// TwinCAT 3 PLC project X881_Booth_Esclave
// libraries:
//   CmpBitmapPool, * (System)
//   Tc2_Standard, * (Beckhoff Automation GmbH)
//   Tc2_SUPS, * (Beckhoff Automation GmbH)
//   Tc2_System, * (Beckhoff Automation GmbH)
//   Tc2_Utilities, * (Beckhoff Automation GmbH)
//   Tc3_Module, * (Beckhoff Automation GmbH)
//   VisuDialogs, * (System)
//   BASIC,3.3.3.0,OSCAT
//   Tc2_ModbusRTU,3.6.1.0,Beckhoff Automation GmbH
//   Tc2_SerialCom,3.4.6.0,Beckhoff Automation GmbH
//   Tc2_SystemCX,3.5.3.0,Beckhoff Automation GmbH
//   Tc2_TcpIp,3.4.2.0,Beckhoff Automation GmbH
//   Util,3.5.11.0,System
//   VisuSymbols,3.5.10.0,System
// project tree:
//   Data types/Autres/ ST_Alarmes.TcDUT
//   Data types/Com_IP/ E_ClientSteps.TcDUT, E_DataExchaSteps.TcDUT, E_ServerSteps.TcDUT
//   Data types/Objets/ Objet_BatElec.TcDUT, Objet_Moteur_EC.TcDUT, Objet_Mot_TOR.TcDUT, Objet_Pressostat.TcDUT, Objet_Registre.TcDUT, Objet_RegulPI.TcDUT, Objet_Sonde.TcDUT
//   Global Variables/ Global_Variables.TcGVL, GVL_RegTROX.TcGVL, GVL_Visu.TcGVL, Variable_Configuration.TcGVL
//   / GlobalTextList.TcGTLO, Recipe Manager.TcRMO (not stored), Standard.TcTTO, Tache_test.TcTTO, Visualization Manager.TcVMO (not stored), VISU_TASK.TcTTO
//   POUs/ a1_MAIN.TcPOU, a2_Gestion_ES.TcPOU, a3_Ecriture_Bit.TcPOU, a4_Lecture_Bit.TcPOU, a5_Ecriture_InterCom.TcPOU, a6_Lecture_InterCom.TcPOU, b_SCL_Mesures.TcPOU, c_Gestion_Defaut.TcPOU, d_Gestion_Pause_Modes.TcPOU, e_Gestion_Horraire.TcPOU, f_Gestion_Etats.TcPOU, g_Gestion_Texte_Modes.TcPOU, h_Enr_Recette.TcPOU, i_Protocol_Auto.TcPOU, j_Protocol_Manu.TcPOU, l_Cons_LED.TcPOU, n0_Regulation_Bas_Deb.TcPOU, n1_Regulation_Press.TcPOU, n2_Regulation_Temp.TcPOU, n3_Regul_Temp_EauMitig.TcPOU, o_Cons_Cmd_Actionneurs.TcPOU, p_Com_Modbus_RS485.TcPOU, q_Gestion_Actionneurs_ANA.TcPOU, r_Gestion_Actionneurs_TOR.TcPOU, s_InterCom_Esclave.TcPOU, t_Enr_Variables.TcPOU
//   POUs/Block/Autres/ Blinck_V2.TcPOU, Dew_Point.TcPOU, Filtre_V1.TcPOU, Prise.TcPOU, PWM.TcPOU, RTC_Time.TcPOU, SCL.TcPOU, SCL_Real.TcPOU, Sontay_4RM.TcPOU, TON_V1.TcPOU, UP_DOWN_RATE.TcPOU
//   POUs/Block/Cabines/ Com485_Dalcnet.TcPOU, Com485_RegTROX.TcPOU, Gache.TcPOU, Humidificateur.TcPOU, Integr_Vol_Eau.TcPOU, Mode.TcPOU, Registre_V1.TcPOU, Servomoteur_V1.TcPOU
//   POUs/Block/Com_Ip/ FB_LocalServer.TcPOU, FB_RemoteClient.TcPOU, FB_ServerDataExcha.TcPOU, LogError.TcPOU, LogMessage.TcPOU, SCODE_CODE.TcPOU
//   POUs/Block/Objets/ BatElec.TcPOU, Moteur_EC.TcPOU, Objet_Mot_TOR_V1.TcPOU, Objet_PI_V1.TcPOU, Objet_Pressostat_V1.TcPOU, Objet_Registre_V1.TcPOU, Objet_Sonde_V1.TcPOU
//   POUs/Gestion_Enceinte_Clim/ B_Gestion_Defaut.TcPOU, C0_Gestion_Consignes.TcPOU, C_Regul_Temp.TcPOU, D_Regul_Humi.TcPOU, E_Cons_Cmd_Actionneurs.TcPOU, F_Gestion_Actionneurs.TcPOU
//   POUs/Visualisation/ Alarmes.TcPOU, Visu.TcPOU
//   Visualizations/Visualizations/ Accueil.TcVIS, Depollution.TcVIS, Maintenance_2.TcVIS, Maintenance_3.TcVIS, Maintenance_4.TcVIS, Maintenance_5.TcVIS, Maintenance_6.TcVIS, Maintenance_7.TcVIS, ModeManuel.TcVIS, Nettoyage.TcVIS, Maintenance_1.TcVIS, menu.TcVIS, Recet_EnCours.TcVIS, Sel_Recettes.TcVIS
//   Visualizations/Visualizations/Fonds/ masque.TcVIS
//   Visualizations/Visualizations/GestionAlarme/Programme/ GestionAlarme.TcPOU
//   Visualizations/Visualizations/GestionAlarme/Structures/ Erreur_Struct.TcDUT, Erreur_StructVisu.TcDUT
//   Visualizations/Visualizations/Images/ ImagePool_Clean.TcIPO (not stored), ImagePool.TcIPO (not stored), ImagePool_Action.TcIPO (not stored), ImagePool_Buttons.TcIPO (not stored)
//   Visualizations/Visualizations/Mes_Textes/ Noms_Modes.TcTLO, Etats_Cabine.TcTLO
//   Visualizations/Visualizations/Objets/ Door.TcVIS, Sink.TcVIS, Drain.TcVIS, Plug.TcVIS
//   Visualizations/Visualizations/PopUp/ Actionneurs.TcVIS, Alarmes.TcVIS, PopUp_Alarms.TcVIS, PopUp_Hight_Level.TcVIS
// real-time tasks:
//   TASK Standard: cycle T#20ms, priority 8, ADS port 350
//   TASK Tache_test: cycle T#10ms, priority 6, ADS port 351
//   TASK VISU_TASK: cycle T#100000us, priority 10, ADS port 352
// I/O:
//   DEVICE Périphérique 2 (EtherCAT), AmsNetId 5.138.94.134.3.1
//     Terme 1 (EK1200) [EK1200-5000 EtherCAT Power supply (2A E-Bus)]
//       Terme 2 (EL1809) [EL1809 16Ch. Dig. Input 24V, 3ms]
//       Terme 3 (EL2828) [EL2828 8Ch. Dig. Output 24V, 2A]
//       Terme 4 (EL3068) [EL3068 8Ch. Ana. Input 0-10V]
//       Terme 5 (EL4008) [EL4008 8Ch. Ana. Output 0-10V, 12bit]
//       Terme 6 (EL6021) [EL6021 Interface (RS422/485)]
//       Terme 7 (EL3068) [EL3068 8Ch. Ana. Input 0-10V]
//       Terme 8 (EL9011) [EL9011 End Terminal]
// variable links:
//   X881_Booth_Esclave/X881_Booth_Esclave Instance <-> Device 2 (EtherCAT)/Term 1 (EK1200)/Term 2 (EL1809)
//     Standard Inputs/Global_Variables.ETOR10_Hygrostat_Souf_CT <-> Channel 10/Input
//     Standard Inputs/Global_Variables.ETOR11_Pressostat_Secu <-> Channel 11/Input
//     Standard Inputs/Global_Variables.ETOR12_Thermostat_Secu <-> Channel 12/Input
//     Standard Inputs/Global_Variables.ETOR13_Marche_BatElec_CTA <-> Channel 13/Input
//     Standard Inputs/Global_Variables.ETOR14_Libre <-> Channel 14/Input
//     Standard Inputs/Global_Variables.ETOR15_Libre <-> Channel 15/Input
//     Standard Inputs/Global_Variables.ETOR16_Libre <-> Channel 16/Input
//     Standard Inputs/Global_Variables.ETOR1_Fdc_Va_Vid_Lavabo_Ouv <-> Channel 1/Input
//     Standard Inputs/Global_Variables.ETOR2_Fdc_Va_Vid_Lavabo_Ferm <-> Channel 2/Input
//     Standard Inputs/Global_Variables.ETOR3_Info_Ma_Prise <-> Channel 3/Input
//     Standard Inputs/Global_Variables.ETOR4_Service_Humi_CTA <-> Channel 4/Input
//     Standard Inputs/Global_Variables.ETOR5_Def_Humi_CTA <-> Channel 5/Input
//     Standard Inputs/Global_Variables.ETOR6_Info_Contact_Porte <-> Channel 6/Input
//     Standard Inputs/Global_Variables.ETOR7_Def_MotRep_Souf_CTA <-> Channel 7/Input
//     Standard Inputs/Global_Variables.ETOR8_Def_MotSouf_Souf_CTA <-> Channel 8/Input
//     Standard Inputs/Global_Variables.ETOR9_Def_Alim_BatElec_CTA <-> Channel 9/Input
//   X881_Booth_Esclave/X881_Booth_Esclave Instance <-> Device 2 (EtherCAT)/Term 1 (EK1200)/Term 3 (EL2828)
//     Standard Outputs/Global_Variables.STOR1_Cmd_EV_Alim_Lavabo <-> Channel 1/Output
//     Standard Outputs/Global_Variables.STOR2_Cmd_Va_Vid_Lavabo <-> Channel 2/Output
//     Standard Outputs/Global_Variables.STOR3_Cmd_Ma_Prise <-> Channel 3/Output
//     Standard Outputs/Global_Variables.STOR4_Cmd_BatElec_CTA <-> Channel 4/Output
//     Standard Outputs/Global_Variables.STOR{5..8}_Libre <-> Channel {5..8}/Output  (4 links)
//   X881_Booth_Esclave/X881_Booth_Esclave Instance <-> Device 2 (EtherCAT)/Term 1 (EK1200)/Term 4 (EL3068)
//     Standard Inputs/Global_Variables.EAN1_Sonde_Debit_Eau_Lavabo <-> AI Standard Channel 1/Value
//     Standard Inputs/Global_Variables.EAN2_Sonde_Temp_Cabine <-> AI Standard Channel 2/Value
//     Standard Inputs/Global_Variables.EAN3_Sonde_Hygro_Cabine <-> AI Standard Channel 3/Value
//     Standard Inputs/Global_Variables.EAN4_Sonde_Temp_Batt_EG <-> AI Standard Channel 4/Value
//     Standard Inputs/Global_Variables.EAN5_Sonde_Pression_Cabine <-> AI Standard Channel 5/Value
//     Standard Inputs/Global_Variables.EAN6_Sonde_press_Souf <-> AI Standard Channel 6/Value
//     Standard Inputs/Global_Variables.EAN7_Retour_Pos_Reg_Etanche_Ext <-> AI Standard Channel 7/Value
//     Standard Inputs/Global_Variables.EAN8_Sonde_press_Ext <-> AI Standard Channel 8/Value
//   X881_Booth_Esclave/X881_Booth_Esclave Instance <-> Device 2 (EtherCAT)/Term 1 (EK1200)/Term 5 (EL4008)
//     Standard Outputs/Global_Variables.SAN1_Cons_Humi_CTA <-> AO Outputs Channel 1/Analog output
//     Standard Outputs/Global_Variables.SAN2_Cons_MotRep_CTA <-> AO Outputs Channel 2/Analog output
//     Standard Outputs/Global_Variables.SAN3_Cons_MotSouf_CTA <-> AO Outputs Channel 3/Analog output
//     Standard Outputs/Global_Variables.SAN4_Cons_BatElec_CTA <-> AO Outputs Channel 4/Analog output
//     Standard Outputs/Global_Variables.SAN5_Cons_V3V_Froid_CTA <-> AO Outputs Channel 5/Analog output
//     Standard Outputs/Global_Variables.SAN6_Libre <-> AO Outputs Channel 6/Analog output
//     Standard Outputs/Global_Variables.SAN8_Libre <-> AO Outputs Channel 8/Analog output
//     Standard Outputs/Global_Variables.SAN7_Cons_Ouv_Reg_Etanche_Ext <-> AO Outputs Channel 7/Analog output
//   X881_Booth_Esclave/X881_Booth_Esclave Instance <-> Device 2 (EtherCAT)/Term 1 (EK1200)/Term 6 (EL6021)
//     Tache_test Inputs/Global_Variables.MB.InData/D[{0..21}] <-> COM TxPDO-Map Inputs/Data In {0..21}  (22 links)
//     Tache_test Inputs/Global_Variables.MB.InData/Status <-> COM TxPDO-Map Inputs/Status
//     Tache_test Outputs/Global_Variables.MB.OutData/Ctrl <-> COM RxPDO-Map Outputs/Ctrl
//     Tache_test Outputs/Global_Variables.MB.OutData/D[{0..21}] <-> COM RxPDO-Map Outputs/Data Out {0..21}  (22 links)
//   X881_Booth_Esclave/X881_Booth_Esclave Instance <-> Device 2 (EtherCAT)/Term 1 (EK1200)/Term 7 (EL3068)
//     Standard Inputs/Global_Variables.EAN{10..16}_Libre <-> AI Standard Channel {2..8}/Value  (7 links)
//     Standard Inputs/Global_Variables.EAN9_Sonde_Temp_Souf <-> AI Standard Channel 1/Value

CONFIGURATION X881_Booth_Esclave
    RESOURCE PLC ON TwinCAT3
        TASK Standard(INTERVAL := T#20ms, PRIORITY := 8);
        TASK Tache_test(INTERVAL := T#10ms, PRIORITY := 6);
        TASK VISU_TASK(INTERVAL := T#100000us, PRIORITY := 10);
        PROGRAM a1_MAIN WITH Standard : a1_MAIN;
        PROGRAM p_Com_Modbus_RS485 WITH Tache_test : p_Com_Modbus_RS485;
        PROGRAM VisuElems_Visu_Prg WITH VISU_TASK : VisuElems.Visu_Prg;
    END_RESOURCE
END_CONFIGURATION

// ---- Data types/Autres/ST_Alarmes.TcDUT
TYPE ST_Alarmes :
STRUCT
	Id          : UINT;          // ID unique
    Libelle     : STRING(80);    // Texte affiché
    Active      : BOOL;          // Vrai si alarme à afficher
END_STRUCT
END_TYPE

// ---- Data types/Com_IP/E_ClientSteps.TcDUT
TYPE E_ClientSteps :
(
	CLIENT_STATE_IDLE,
	CLIENT_STATE_CONNECT_START,
	CLIENT_STATE_CONNECT_WAIT,
	CLIENT_STATE_DATAEXCHA_START,
	CLIENT_STATE_DATAEXCHA_WAIT,
	CLIENT_STATE_CLOSE_START,
	CLIENT_STATE_CLOSE_WAIT,
	CLIENT_STATE_ERROR
);
END_TYPE

// ---- Data types/Com_IP/E_DataExchaSteps.TcDUT
TYPE E_DataExchaSteps :
(
	DATAEXCHA_STATE_IDLE,
	DATAEXCHA_STATE_SEND_START,
	DATAEXCHA_STATE_SEND_WAIT,
	DATAEXCHA_STATE_RECEIVE_START,
	DATAEXCHA_STATE_RECEIVE_WAIT,
	DATAEXCHA_STATE_ERROR
);
END_TYPE

// ---- Data types/Com_IP/E_ServerSteps.TcDUT
TYPE E_ServerSteps :
(
	SERVER_STATE_IDLE,
	SERVER_STATE_LISTENER_OPEN_START,
	SERVER_STATE_LISTENER_OPEN_WAIT,
	SERVER_STATE_REMOTE_CLIENTS_COMM,
	SERVER_STATE_REMOTE_CLIENTS_CLOSE,
	SERVER_STATE_LISTENER_CLOSE_START,
	SERVER_STATE_LISTENER_CLOSE_WAIT,
	SERVER_STATE_ERROR
);
END_TYPE

// ---- Data types/Objets/Objet_BatElec.TcDUT
TYPE Objet_BatElec :
	STRUCT
		Mot_Lecture 				:INT; (*Mot de lecture des bits*)
		Mot_Ecriture 				:INT; (*Mot d'écriture des bits*)
		R_TempApresBat			: REAL; (* en °C *)
		R_Info_Cons				: REAL; (* en % *)
		W_LimiteMinCons			: REAL; (* en % *)
		W_LimiteMaxCons 		: REAL; (* en % *)
		W_ConsForcage			: REAL; (* en % *)
		W_SeuilTempMax			: REAL; (* en °C *)
		W_PeriodePWM			: REAL; (* en sec *)
		W_TempsMinPWM		: REAL; (* en sec *)
		W_TempsMaxPWM		: REAL; (* en sec *)
	END_STRUCT
END_TYPE

// ---- Data types/Objets/Objet_Moteur_EC.TcDUT
TYPE Objet_Moteur_EC :
	STRUCT
	Mot_Lecture 			:INT; (*Mot de lecture des bits*)
	Mot_Ecriture 			:INT; (*Mot d'écriture des bits*)
	R_LimiteMinFreq 		:REAL; (*Info Limite basse vitesse*)
	R_LimiteMaxFreq 		:REAL; (*Info Limite haute vitesse*)
	R_InfoFreq			:REAL; (*Mesure de la vitesse*)
	R_InfoCons 			:REAL; (*Info consigne appliquée*)
	W_LimiteMinCons 		:REAL; (*Consigne limite basse*)
	W_LimiteMaxCons 	:REAL; (*Consigne limite haute*)
	W_ConsOccupe 		:REAL; (*Consigne mode occupé*)
	W_ConsInoccupe 		:REAL; (*Consigne mode inoccupé*)
	W_ConsForcage 		:REAL; (*Consigne mode forcé*)
	END_STRUCT
END_TYPE

// ---- Data types/Objets/Objet_Mot_TOR.TcDUT
TYPE Objet_Mot_TOR :
STRUCT
		Mot_Lecture 	:INT; (*Mot de lecture des bits*)
		Mot_Ecriture 	:INT; (*Mot d'écriture des bits*)
END_STRUCT
END_TYPE

// ---- Data types/Objets/Objet_Pressostat.TcDUT
TYPE Objet_Pressostat :
STRUCT
	Mot_Lecture 			:INT; (*Mot de lecture des bits*)
	Mot_Ecriture 			:INT; (*Mot d'écriture des bits*)
	R_SeuilPress	 		:REAL; (* en Pa *)
END_STRUCT
END_TYPE

// ---- Data types/Objets/Objet_Registre.TcDUT
TYPE Objet_Registre :
STRUCT
	Mot_Lecture 			:INT; (*Mot de lecture des bits*)
	Mot_Ecriture 			:INT; (*Mot d'écriture des bits*)
	R_InfoConsPosition	: REAL; (* en % *)
	R_Position			: REAL; (* en % *)
	W_ConsForcage		: REAL; (* en % *)
	W_LimiteMinPosition	: REAL; (* en % *)
	W_LimiteMaxPosition 	: REAL; (* en % *)
END_STRUCT
END_TYPE

// ---- Data types/Objets/Objet_RegulPI.TcDUT
TYPE Objet_RegulPI :
STRUCT
	Mot_Lecture 			:INT; (*Mot de lecture des bits*)
	Mot_Ecriture 			:INT; (*Mot d'écriture des bits*)
	R_InfoConsPI			: REAL; (* L'unité dépend de la régulation (°C / % / Pa / bar / m3/h / mg/l ect ....) *)
	R_MesRegulPI		: REAL; (* L'unité dépend de la régulation (°C / % / Pa / bar / m3/h / mg/l ect ....) *)
	R_SortieCmdPI		: REAL; (* L'unité dépend de la régulation (°C / % / Pa / bar / m3/h / mg/l ect ....) *)
	W_ConsOccupe		: REAL; (* L'unité dépend de la régulation (°C / % / Pa / bar / m3/h / mg/l ect ....) *)
	W_ConsInoccupe		: REAL; (* L'unité dépend de la régulation (°C / % / Pa / bar / m3/h / mg/l ect ....) *)
	W_ConsPIForcage	: REAL; (* en °C *)
	W_LimiteMinCons		: REAL; (* L'unité dépend de la régulation (°C / % / Pa / bar / m3/h / mg/l ect ....) *)
	W_LimiteMaxCons 	: REAL; (* L'unité dépend de la régulation (°C / % / Pa / bar / m3/h / mg/l ect ....) *)
	W_GainPI 			: REAL; (* en % *)
	W_IntegralPI 			: REAL; (* en sec *)
	W_DerivPI 			: REAL; (* en sec *)
	W_BandeMorte		: REAL; (* L'unité dépend de la régulation (°C / % / Pa / bar / m3/h / mg/l ect ....) *)
	W_SortieCMDForcage	: REAL; (* L'unité dépend de la régulation (°C / % / Pa / bar / m3/h / mg/l ect ....) *)
END_STRUCT
END_TYPE

// ---- Data types/Objets/Objet_Sonde.TcDUT
TYPE Objet_Sonde :
	STRUCT
	Mot_Lecture 			:INT; (*Mot de lecture des bits*)
	Mot_Ecriture 			:INT; (*Mot d'écriture des bits*)
	R_MesBrut 			:REAL; (*Mesure de la température brute*)
	R_MesCor 			:REAL; (*Mesure de la température corrigée*)
	W_Offset				:REAL; (* Consigne Offset de température*)
	W_SeuilAlarmeHaute 	:REAL; (*Consigne du seuil haut du déclenchement de l'alarme haute température*)
	W_SeuilAlarmeBasse 	:REAL; (*Consigne du seuil bas du déclenchement de l'alarme basse température*)
	END_STRUCT
END_TYPE

// ---- Visualizations/Visualizations/GestionAlarme/Structures/Erreur_Struct.TcDUT
TYPE Erreur_Struct :
STRUCT
	IdDefaut : INT; //Identifiant dans la text list
	DateDefaut : STRING; //Heure d'arrivé du défaut
	TypeDefaut : SINT ; //0=Erreur;1=Warning;2=Warning acquittable	
	EtatDefaut : STRING(3); //DP = Defaut présent; DD = Defaut disparu non acquité ; WP = warning présent ; WD = Warning disparu non acquité; WA = Warning aquittable
END_STRUCT
END_TYPE

// ---- Visualizations/Visualizations/GestionAlarme/Structures/Erreur_StructVisu.TcDUT
TYPE Erreur_StructVisu :
STRUCT
	TypeDefaut : STRING(3);
	IDMessage : INT;
	DateMessage : STRING(200);
END_STRUCT
END_TYPE

// ---- Global Variables/Global_Variables.TcGVL
//{attribute 'Tc2GvlVarNames'}Tc2GvlVarNames
 VAR_GLOBAL
(* Configuration des E/S *)
	ETOR1_Fdc_Va_Vid_Lavabo_Ouv			AT %IX0.0 : BOOL;
	ETOR2_Fdc_Va_Vid_Lavabo_Ferm		AT %IX0.1 : BOOL;
	ETOR3_Info_Ma_Prise					AT %IX0.2 : BOOL;
	ETOR4_Service_Humi_CTA				AT %IX0.3 : BOOL;
	ETOR5_Def_Humi_CTA					AT %IX0.4 : BOOL;
	ETOR6_Info_Contact_Porte			AT %IX0.5 : BOOL;
	ETOR7_Def_MotRep_Souf_CTA			AT %IX0.6 : BOOL;
	ETOR8_Def_MotSouf_Souf_CTA 			AT %IX0.7 : BOOL;
	ETOR9_Def_Alim_BatElec_CTA			AT %IX0.8 : BOOL;
	ETOR10_Hygrostat_Souf_CT			AT %IX0.9:BOOL;
	ETOR11_Pressostat_Secu				AT %IX0.10:BOOL;
	ETOR12_Thermostat_Secu				AT %IX0.11: BOOL;
	ETOR13_Marche_BatElec_CTA			AT %IX0.12: BOOL;
	ETOR14_Libre 						AT %IX0.13 : BOOL;
	ETOR15_Libre 						AT %IX0.14 : BOOL;
	ETOR16_Libre 						AT %IX0.15 : BOOL;

	STOR1_Cmd_EV_Alim_Lavabo			AT %QX0.0 : BOOL;
	STOR2_Cmd_Va_Vid_Lavabo				AT %QX0.1 : BOOL;
	STOR3_Cmd_Ma_Prise					AT %QX0.2 : BOOL;
	STOR4_Cmd_BatElec_CTA				AT %QX0.3 : BOOL;
	STOR5_Libre							AT %QX0.4: BOOL;
	STOR6_Libre							AT %QX0.5: BOOL;
	STOR7_Libre							AT %QX0.6: BOOL;
	STOR8_Libre							AT %QX0.7: BOOL;

	EAN1_Sonde_Debit_Eau_Lavabo	 		AT %I* : INT;
	EAN2_Sonde_Temp_Cabine 				AT %I* : INT;
	EAN3_Sonde_Hygro_Cabine				AT %I* : INT;
	EAN4_Sonde_Temp_Batt_EG				AT %I* : INT;
	EAN5_Sonde_Pression_Cabine			AT %I* : INT;
	EAN6_Sonde_press_Souf				AT %I* : INT;
	EAN7_Retour_Pos_Reg_Etanche_Ext		AT %I* : INT;
	EAN8_Sonde_press_Ext				AT %I* : INT;
	
	EAN9_Sonde_Temp_Souf		 		AT %I* : INT;
	EAN10_Libre							AT %I* : INT;
	EAN11_Libre							AT %I* : INT;
	EAN12_Libre							AT %I* : INT;
	EAN13_Libre							AT %I* : INT;
	EAN14_Libre							AT %I* : INT;
	EAN15_Libre							AT %I* : INT;
	EAN16_Libre							AT %I* : INT;

	SAN1_Cons_Humi_CTA					AT %Q*:INT;
	SAN2_Cons_MotRep_CTA 				AT %Q*:INT;
	SAN3_Cons_MotSouf_CTA				AT %Q*:INT;
	SAN4_Cons_BatElec_CTA				AT %Q*:INT;
	SAN5_Cons_V3V_Froid_CTA				AT %Q*:INT;
	SAN6_Libre							AT %Q*:INT;
	SAN7_Cons_Ouv_Reg_Etanche_Ext		AT %Q*:INT;
	SAN8_Libre							AT %Q*:INT;

	MB : ModbusRtuMaster_KL6x22B;

(******************************************************************************************)
(*Gestion Intercommunication entre automate*)
(*****************Com IP gestion option automate esclave*************************)
	bLogDebugMessages					: BOOL := TRUE;
	MAX_CLIENT_CONNECTIONS				: UDINT(1..20) := 1;
	MAX_PLCPRJ_RXBUFFER_SIZE			: UDINT := 1000;
	PLCPRJ_RECONNECT_TIME				: TIME := T#3S;
(*	PLCPRJ_SEND_CYCLE_TIME				: TIME := T#1s; not used at server side *)
	PLCPRJ_ACCEPT_POLLING_TIME			: TIME := T#1S;
	PLCPRJ_RECEIVE_POLLING_TIME		 	: TIME := T#1S;
	PLCPRJ_RECEIVE_TIMEOUT				: TIME := T#50S;
	(* Some project specific error codes *)
	PLCPRJ_ERROR_RECEIVE_BUFFER_OVERFLOW	: UDINT := 16#8101; (* receive buffer overflow*)
	PLCPRJ_ERROR_RECEIVE_TIMEOUT		: UDINT := 16#8102;(* receive timeout error *)
	Tab_Com_Send						: ARRAY [0..30] OF REAL;
	Tab_Com_Receive						: ARRAY [0..30] OF REAL;
	fbServer							: FB_LocalServer;

(************Gestion ecriture Inter-com Cabine************)
	Temperature_Cabine 					:REAL;
	Hygrometrie_Cabine 					:REAL;
	(*à définir en focntion de la gestion de l'automate maître*)

(************Gestion lecture Inter-com Cabine************)
	(*à définir en focntion de la gestion de l'automate maître*)
	Van_Maitre							:WORD;
	Vmois_Maitre						:WORD;
	Vjour_Maitre						:WORD;
	Vheure_Maitre						:WORD;
	Vminute_Maitre						:WORD;
	VDayOfWeek_Maitre					:WORD;

(******************************************************************************************)
(*GESTION DES VARIABLES DE LA CABINE*)
(******************************************************************************************)

(*Autres (Non utilisé dans la table d'échange)*)
	(*Gestion des états*)
	Mode_Occupation						: BOOL;
	Mode_Evaluation						: BOOL;
	Mode_Neutre							: BOOL;
	Arret_Extraction					: BOOL;
	Arret_Soufflage						: BOOL;
	Arret_Petit_Debit					: BOOL;
	Defaut_General_Alim_Eau				: BOOL;
	Mode_Depollution_cycle1				: BOOL;
	(*Gestion error com modebus RS485*)
	Temp_Eau_Mitige						: INT;
	Temp_Cons_Eau_Mitige				: INT;
	Com_Ok_Dalcnet						: BOOL;
	Error_Dalcnet						: BOOL;
	Com_Ok_Vanne_Thermo					: BOOL;
	Error_Vanne_Thermo					: BOOL;
 	(*Calcul des ecart de régulations*)
	S_Ecart_Regul_PID_Extraction		: REAL;
	S_Ecart_Regul_PID_Soufflage			: REAL;
	S_Ecart_Regul_PID_Pression			: REAL;
	S_Ecart_Regul_PID_Temp_Eau_Mitig	: REAL;
	(*Gestion des recettes auto et manu*)
	Mode_Auto							: Mode;
	Mode_Manu							: Mode;
	(*Alarme qui met en pause les recettes*)
	Alarme_Secu_Mode_1					: BOOL;
	Alarme_Secu_Mode_2					: BOOL;
	Alarme_Secu_Mode_3					: BOOL;
	Alarme_Secu_Mode_4					: BOOL;
	Alarme_Secu_Mode_5					: BOOL;
	Alarme_Secu_Mode_6					: BOOL;
	Alarme_Secu_Mode_7					: BOOL;
	Alarme_Secu_Mode_8					: BOOL;
	Alarme_Secu_Mode_10					: BOOL;
	Alarme_Secu_Mode_11					: BOOL;
	Alarme_Secu_Mode_12					: BOOL;
	Alarme_Secu_Mode_13					: BOOL;
	Alarme_Secu_Mode_14					: BOOL;
	Alarme_Secu_Mode_15					: BOOL;
	Alarme_Secu_Mode_16					: BOOL;
	Alarme_Secu_Mode_17					: BOOL;
	Alarme_Secu_Mode_18					: BOOL;
	Alarme_Secu_Mode_19					: BOOL;
	Alarme_Secu_Mode_23					: BOOL;
	Alarme_Secu_Mode_24					: BOOL;
	(*Horodatage*)
	Van 								: WORD; (* Année courante *)
	Vmois								: WORD; (* Mois courante *)
	Vjour								: WORD; (* Jour courante *)
	Vheure								: WORD; (* Heure courante *)
	Vminute								: WORD; (* Minute courante *)
	Vseconde							: WORD; (* Seconde courante *)
	VDayOfWeek							: WORD; (* Jour de la semaine *)
	(*Gestion mode arrêt des modes manu et auto*)
	Mode_Arret_Manu 					:BOOL;
	Mode_Arret_Auto 					:BOOL;
	Mode_Warning						:BOOL;
	(*etape du de l'éxécution du mode auto et manu*)
	Numero_Mode_Auto					: INT;
	Numero_Mode_Manu					: INT;
	(*Lecture commande et consigne actionneur*)
	Cmd_Appli_PC_Cab 					: BOOL;
	Cmd_Appli_Vanne_Alim_Douche 		: BOOL;
	Cmd_Appli_Vanne_Alim_Douchette 		: BOOL;
	Cmd_Appli_Vanne_Alim_NEP 			: BOOL;
	Cmd_Appli_Vanne_Alim_Lavabo 		: BOOL;
	Cmd_Appli_Vanne_Vid_Douche 			: BOOL;
	Cmd_Appli_Vanne_Vid_Lavabo 			: BOOL;
	Cmd_Appli_ElectroValve_Alim_Douche 	: BOOL;
	Cmd_Appli_ElectroValve_Alim_Lavabo 	: BOOL;
	Cmd_Appli_BattElec 					:BOOL;
	Cons_Temperature_Eau_F				: INT;
	Cmd_Appli_Vanne_Souf_Bas_Deb 		:BOOL;
	Cmd_Appli_Vanne_Ext_Bas_Deb 		:BOOL;
	Cmd_Appli_Reg_Etanche_Souf 			:BOOL;
	Cmd_Appli_Verin_WC_GV				: BOOL;
	Cmd_Appli_Verin_WC_PV				: BOOL;
	(*Variable PID*)
	Enable_PID_Bas_Deb_Ext				: BOOL;
	S_Cmd_PID_Bas_Deb_Ext				: REAL;
	Enable_PID_Temp_Amb					: BOOL;
	S_Cmd_PID_Temp_Amb					: REAL;
	Enable_PID_Press_Cab				: BOOL;
	S_Cmd_PID_Press_Cab					: REAL;
	Enable_PID_Temp_Eau_Mitig			: BOOL;
	S_Cmd_PID_Temp_Eau_Mitig			: REAL;
	Regul_Humi_YMin						: REAL;
	(*Temporisation de sécurisation des alimentations*)
	Temp_Secu_Debord_Douche_Int			: INT;
	Temp_Secu_Debord_Lavabo_Int			: INT;
	Mes_Out_Max							: REAL;
	Forc_Ouv_Alim_Lav_Dou				: BOOL;
	FCV_01_extraction					: Registre_V1;
	FCV_02_soufflage					: Registre_V1;
	(*Gestion des mesures*)
	E_Sonde_Gros_Debit_Soufflage_1 		:INT;
	E_Sonde_Gros_Debit_Extraction_1 	:INT;
	(*Option non utilisé*)
	Option_Vanne_Thermo_General 		: BOOL;
	Option_Vanne_Thermo_Par_Cabine 		: BOOL;

(**********************************************************************************************)
(*configuration des Entrees tor et ana*)
	E_Info_Niveau_Haut_Douche			: BOOL;
	E_Info_Niveau_Haut_Lavabo 			: BOOL;
	E_Info_Contact_Porte 				: BOOL;
	E_Info_PC_Cab 						: BOOL;
	E_Etat_Evac_SaniDouche 				: BOOL;
	E_Info_Klixon_BattElec 				:BOOL;
	E_Defaut_Prise_Elec 				:BOOL;

	E_Vanne_Alim_Douche_Ouv 			: BOOL;
	E_Vanne_Alim_Douche_Ferm 			: BOOL;
	E_Vanne_Alim_Douchette_Ouv 			: BOOL;
	E_Vanne_Alim_Douchette_Ferm 		: BOOL;
	E_Vanne_Alim_Lavabo_Ouv 			: BOOL;
	E_Vanne_Alim_Lavabo_Ferm 			: BOOL;
	E_Vanne_Vidange_Douche_Ouv 			: BOOL;
	E_Vanne_Vidange_Douche_Ferm 		: BOOL;
	E_Vanne_Vidange_Lavabo_Ouv 			: BOOL;
	E_Vanne_Vidange_Lavabo_Ferm 		: BOOL;
	E_Vanne_Alim_NEP_Ouv 				:BOOL;
	E_Vanne_Alim_NEP_Ferm 				:BOOL;

	E_Vanne_Souf_Bas_Deb_Ouv 			:BOOL;
	E_Vanne_Souf_Bas_Deb_Ferm 			:BOOL;
	E_Vanne_Ext_Bas_Deb_Ouv 			:BOOL;
	E_Vanne_Ext_Bas_Deb_Ferm 			:BOOL;

	E_Sonde_Temp_Amb 					: INT;
	E_Sonde_Hygro_Amb 					: INT;
	E_Sonde_Pression_Cabine 			:INT;
	E_Sonde_Temp_Eau_Mitig 				:INT;
	E_Sonde_press_Souf 					:INT;
	E_Sonde_press_Ext 					:INT;
	E_Sonde_Temp_Batt_EG 				:INT;

	E_Sonde_Gros_Debit_Soufflage 		: INT;
	E_Sonde_Gros_Debit_Extraction 		: INT;
	E_Sonde_Petit_Debit_Extraction 		: INT;
	E_Sonde_Pression_ByPass 			:INT;
	E_Retour_Pos_Reg_Etanche_Ext 		:INT;

	E_Sonde_Debit_Alim_Douche 			:INT;
	E_Sonde_Debit_Alim_Lavabo 			:INT;
	E_Sonde_Temp_Souf					:INT;
(*Sorties tor et ana*)
	S_Cmd_PC_Cab 						: BOOL;
	S_Cmd_Vanne_Alim_Douche 			: BOOL;
	S_Cmd_Vanne_Alim_Douchette 			: BOOL;
	S_Cmd_Vanne_Alim_Lavabo 			: BOOL;
	S_Cmd_Vanne_Vid_Douche 				: BOOL;
	S_Cmd_Vanne_Vid_Lavabo 				: BOOL;
	S_Cmd_ElectroValve_Alim_Douche 		: BOOL;
	S_Cmd_ElectroValve_Alim_Lavabo 		: BOOL;
	S_Cmd_BattElec 						:BOOL;
	S_Cmd_Vanne_Souf_Bas_Deb 			:BOOL;
	S_Cmd_Vanne_Ext_Bas_Deb 			:BOOL;
	S_Cmd_Reg_Etanche_Souf 				:BOOL;
	S_Cmd_Vanne_NEP 					: BOOL;
	S_Cmd_Appli_Verin_WC_GV				: BOOL;
	S_Cmd_Appli_Verin_WC_PV				: BOOL;

	S_Cons_Registre_Extraction 			: INT;
	S_Cons_Registre_Soufflage 			: INT;
	S_Cons_Moteur_BasDebit 				: INT;
	S_Cons_Moteur_ByPass				: INT;
	S_Cons_BattElec 					:INT;
	S_Cons_Reg_Etanche_Ext 				:INT;
	S_Cons_Ouv_V3V_Eau_Mitig 			:INT;
	S_Cons_Module_Sontay 				:INT;

(*Configuration des Entrées et Sorties - Gestion des enceintes climatiques*)
	E_Def_MotRep_CTA 					: BOOL;
	E_Def_MotSouf_CTA 					: BOOL;
	E_Hygrostat_Souf_CTA 				: BOOL;
	E_Def_Alim_BatElec_CTA				: BOOL;
	E_Marche_BatElec_CTA 				: BOOL;
	E_Def_Humi_CTA 						: BOOL;
	E_Service_Humi_CTA 					: BOOL;
	E_Pressostat_Secu 					: BOOL;
	E_Thermostat_Secu 					: BOOL;

	S_Cmd_BatElec_CTA 					: BOOL;
	S_Cmd_Humi_CTA 						: BOOL;

	S_Cons_V3V_Froid_CTA				:INT;
	S_Cons_MotRep_CTA 					:INT;
	S_Cons_MotSouf_CTA 					:INT;
	S_Cons_BatElec_CTA 					:INT;
	S_Cons_Humi_CTA 					:INT;

(*Gestion des alarmes*)
	(*Non récupérer sur GTC*)
	Securite_Debord_Douche 				:BOOL;
	Securite_Debord_Lavabo 				:BOOL;
	(*Défaut récupéré sur GTC*)
	Defaut_Debordement_Douche			: BOOL;
	Defaut_Debordement_Lavabo			: BOOL;
	Defaut_Discord_Deb_Eau_Douche 		:BOOL;
	Defaut_Discord_Deb_Eau_Lavabo		 :BOOL;

	Defaut_Discord_PC_Cab				: BOOL;
	Def_Discord_Alim_Prise				: BOOL;
	Def_Prise_Porte_Ouverte				: BOOL;
	Defaut_Pompe_Relevage				: BOOL;
	Defaut_Porte_Ouverte				: BOOL;

	Defaut_Com_Dalcnet					: BOOL;
	Defaut_Com_Vanne_Thermo 			:BOOL;
	Defaut_Com_Vanne_General 			:BOOL;
	Defaut_Com_Client					:BOOL;

	Defaut_Discord_Vanne_Vid_Douche_Ouv		: BOOL;
	Defaut_Discord_Vanne_Vid_Douche_Ferm	: BOOL;
	Defaut_Discord_Vanne_Vid_Lavabo_Ouv		: BOOL;
	Defaut_Discord_Vanne_Vid_Lavabo_Ferm	: BOOL;
	Defaut_Discord_Vanne_Alim_Douche_Ouv	: BOOL;
	Defaut_Discord_Vanne_Alim_Douche_Ferm	: BOOL;
	Defaut_Discord_Vanne_Alim_Lavabo_Ouv	: BOOL;
	Defaut_Discord_Vanne_Alim_Lavabo_Ferm	: BOOL;
	Defaut_Discord_Vanne_Alim_Douchette_Ouv	: BOOL;
	Defaut_Discord_Vanne_Alim_Douchette_Ferm: BOOL;
	Defaut_Discord_Vanne_Alim_NEP_Ouv		: BOOL;
	Defaut_Discord_Vanne_Alim_NEP_Ferm		: BOOL;

	Defaut_Discord_Vanne_Souf_Bas_Deb_Ouv 	:BOOL;
	Defaut_Discord_Vanne_Souf_Bas_Deb_Ferm 	:BOOL;
	Defaut_Discord_Vanne_Ext_Bas_Deb_Ouv 	:BOOL;
	Defaut_Discord_Vanne_Ext_Bas_Deb_Ferm 	:BOOL;

	Defaut_Discord_Deb_Ext				: BOOL;
	Defaut_Discord_Deb_Souf				: BOOL;
	Defaut_Discord_Reg_Souf_Ferm		: BOOL;
	Defaut_Discord_Reg_Ext_Ferm			: BOOL;
	Defaut_Klixon_BattElec				: BOOL;

	Defaut_Discord_Reg_Etanche_Ext 		:BOOL;
	Defaut_Discord_Regul_Press_Cab 		:BOOL;
	Defaut_Differentiel_Prise_Elec 		:BOOL;
	Defaut_Com_Reg_Souf 				:BOOL;
	Defaut_Com_Reg_Ext 					:BOOL;
	Defaut_Ensemble_Bas_Debit 			:BOOL;
	Defaut_Ensemble_Bypass 				:BOOL;
	Defaut_Sonde_Press_Cabine 			:BOOL;
	Defaut_Sonde_Temp_Cabine 			:BOOL;
	Defaut_Sonde_Hygro_Cabine 			:BOOL;
	Defaut_Sonde_Temp_Eau_Mitig 		:BOOL;
	
	Defaut_Sonde_Temp_Souf				:BOOL;

(*Bit lecture gestion recette et état de la cabine*)
	Mode_Cabine_Eclairage				: BOOL;
	Mode_Cabine_Defaut					: BOOL;
	Mode_Cabine_Libre					: BOOL;
	Mode_Cabine_Manuel					: BOOL;
	Mode_Cabine_Automatique				: BOOL;
	Mode_Cabine_Depollution				: BOOL;
	Mode_Cabine_Nettoyage				: BOOL;
	Mode_Maintenance					: BOOL;

	Statut_Pause_Force					: BOOL;
	Attente_Reset_Pause					: BOOL;
	Comande_Pause						: BOOL;
	Condi_Affich_Etape_Suiv				: BOOL;
	Condi_Affich_Rearm					: BOOL;

(*Lecture des consignes appliquée (Sortie bloc mode)*)
	(*Affichage du texte du mode en cours*)
	Lecture_Texte_Choisi_FR				AT %MW1: STRING(139); (*Adresse Modbus GTC : 12289*)
	Lecture_Texte_Choisi_ENG			AT %MW71: STRING(139); (*Adresse Modbus GTC : 12359*)

(*étape et états de la cabine*)
	Sel_Etats_Cabine 					AT %MW7211: INT; (*Adresse Modbus GTC : 19499*)
	Nbre_Etape_Totale 					AT %MW7212: INT; (*Adresse Modbus GTC : 19500*)
	Numero_Etape_Actuel 				AT %MW7213: INT; (*Adresse Modbus GTC : 19501*)

(* Gestion de la lumière en lecture*)
	Cde_Dimmer_Cabine					AT %MW7214: INT; (*Adresse Modbus GTC : 19502*)
	Cde_Rouge_Cabine					AT %MW7215: INT; (*Adresse Modbus GTC : 19503*)
	Cde_Vert_Cabine						AT %MW7216: INT; (*Adresse Modbus GTC : 19504*)
	Cde_Bleu_Cabine						AT %MW7217: INT; (*Adresse Modbus GTC : 19505*)
	Cde_Blanc_Cabine					AT %MW7218: INT; (*Adresse Modbus GTC : 19506*)

(*Lecture des consignes appliquée (Sortie bloc mode)*)
	(*Décompte de la temporisation et visualisation du volume d'eau*)
	Temp_Restant_Seconde				AT %MW7220: REAL; (*Adresse Modbus GTC : 19508*)
	Temp_Restant_Minute					AT %MW7222: REAL; (*Adresse Modbus GTC : 19510*)
	Temp_Restant_Heure					AT %MW7224: REAL; (*Adresse Modbus GTC : 19512*)
	Lect_Volume_Eau_Douche				AT %MW7226: REAL; (*Adresse Modbus GTC : 19514*)
	Lect_Volume_Eau_Lavabo				AT %MW7228: REAL; (*Adresse Modbus GTC : 19516*)
	(*Consigne de ventilation et consigne de température d'eau*)
	Cons_Deb_Soufflage_Appli			AT %MW7230: REAL; (*Adresse Modbus GTC : 19518*)
	Cons_Deb_Extraction_Appli			AT %MW7232: REAL; (*Adresse Modbus GTC : 19520*)
	Cons_Temperature_Eau_Appli			AT %MW7234: REAL; (*Adresse Modbus GTC : 19522*)
	Cons_Para_Nbre_Chasse_Eau			AT %MW7236: REAL; (*Adresse Modbus GTC : 19524*)
	Cons_Para_11_Appli					AT %MW7238: REAL; (*Adresse Modbus GTC : 19526*)
	Cons_Para_12_Appli					AT %MW7240: REAL; (*Adresse Modbus GTC : 19528*)
	Cons_Para_13_Appli					AT %MW7242: REAL; (*Adresse Modbus GTC : 19530*)
	Cons_Para_14_Appli					AT %MW7244: REAL; (*Adresse Modbus GTC : 19532*)
	Cons_Para_15_Appli					AT %MW7246: REAL; (*Adresse Modbus GTC : 19534*)
	(*Gestion du décompte du nombre de chasse*)
	Nbre_Chasse_Total					AT %MW9814: REAL; (*Adresse Modbus GTC : 22102*)
	Nbre_Chasse_EnCours					AT %MW9816: REAL; (*Adresse Modbus GTC : 22104*)

(*Lecture des consignes actuel (Entrée bloc mode)*)
	Numero_Mode_Actuel					AT %MW7248: REAL; (*Adresse Modbus GTC : 19536*)
	Tempo_Transition_seconde_Actuel		AT %MW7250: REAL; (*Adresse Modbus GTC : 19538*)
	Tempo_Transition_Minute_Actuel		AT %MW7252: REAL; (*Adresse Modbus GTC : 19540*)
	Tempo_Transition_Heure_Actuel		AT %MW7254: REAL; (*Adresse Modbus GTC : 19542*)

	Cons_Volume_Eau_Douche_Actuel		AT %MW7256: REAL; (*Adresse Modbus GTC : 19544*)
	Cons_Volume_Eau_Lavabo_Actuel		AT %MW7258: REAL; (*Adresse Modbus GTC : 19546*)
	Cons_Deb_Soufflage_Actuel			AT %MW7260: REAL; (*Adresse Modbus GTC : 19548*)
	Cons_Deb_Extraction_Actuel			AT %MW7262: REAL; (*Adresse Modbus GTC : 19550*)
	Cons_Temperature_Eau_Actuel			AT %MW7264: REAL; (*Adresse Modbus GTC : 19552*)
	Cons_Para_10_Actuel					AT %MW7266: REAL; (*Adresse Modbus GTC : 19554*)
	Cons_Para_11_Actuel					AT %MW7268: REAL; (*Adresse Modbus GTC : 19556*)
	Cons_Para_12_Actuel					AT %MW7270: REAL; (*Adresse Modbus GTC : 19558*)
	Cons_Para_13_Actuel					AT %MW7272: REAL; (*Adresse Modbus GTC : 19560*)
	Cons_Para_14_Actuel					AT %MW7274: REAL; (*Adresse Modbus GTC : 19562*)
	Cons_Para_15_Actuel					AT %MW7276: REAL; (*Adresse Modbus GTC : 19564*)

(*Mesures*)
	MES_Debit_Volh_Extraction 			AT %MW7278: REAL; (*Adresse Modbus GTC : 19566*)
	MES_Debit_Volh_Soufflage 			AT %MW7280: REAL; (*Adresse Modbus GTC : 19568*)
	MES_Petit_Debit_Volh_Extraction 	AT %MW7282: REAL; (*Adresse Modbus GTC : 19570*)	
	MES_Petit_Debit_m3h_Extraction		AT %MW7316: REAL; (*Adresse Modbus GTC : 19604*)	
	MES_Sonde_Temp_Amb_F				AT %MW7284: REAL; (*Adresse Modbus GTC : 19572*)
	MES_Temp_Eau_Mitige_Cabine			AT %MW7286: REAL; (*Adresse Modbus GTC : 19574*)
	MES_Temp_Eau_Mitige_Cabine_F		AT %MW7288: REAL; (*Adresse Modbus GTC : 19576*)
	MES_Temp_Eau_Mitige_General			AT %MW7290: REAL; (*Adresse Modbus GTC : 19578*)
	MES_Temp_Eau_Mitige_General_F		AT %MW7292: REAL; (*Adresse Modbus GTC : 19580*)	
	MES_Debit_ByPass_Volh				AT %MW9050: REAL; (*Adresse Modbus GTC : 21338*)
	MES_Debit_ByPass_m3h				AT %MW9052: REAL; (*Adresse Modbus GTC : 21340*)
	MES_Pos_Reg_Etanche_Ext				AT %MW9054: REAL; (*Adresse Modbus GTC : 21342*)	
	MES_Pos_Reg_Souf					AT %MW9076: REAL; (*Adresse Modbus GTC : 21364*)

(*Lectures des consignes Actionneur*)
	Cons_Actionneur_Registre_Ext_Volh 	AT %MW7294: REAL; (*Adresse Modbus GTC : 19582*)
	Cons_Actionneur_Registre_Souf_Volh 	AT %MW7296: REAL; (*Adresse Modbus GTC : 19584*)
	Cons_Actio_Registre_Ext_m3h			AT %MW7298: REAL; (*Adresse Modbus GTC : 19586*)
	Cons_Actio_Registre_Souf_m3h 		AT %MW7300: REAL; (*Adresse Modbus GTC : 19588*)
	Cons_Actionneur_Moteur_BasDebit 	AT %MW7302: REAL; (*Adresse Modbus GTC : 19590*)
	Cons_Actionneur_Moteur_ByPass		AT %MW7304: REAL; (*Adresse Modbus GTC : 19592*)
	Cons_Actionneur_BattElec			AT %MW7306: REAL; (*Adresse Modbus GTC : 19594*)
	Cons_Temperature_Eau				AT %MW7308: REAL; (*Adresse Modbus GTC : 19596*)
	
	Cons_Actionneur_Reg_Etanche_Ext 	AT %MW9056: REAL; (*Adresse Modbus GTC : 21344*)
	Cons_Actionneur_V3V_Eau_Mitig		AT %MW9058: REAL; (*Adresse Modbus GTC : 21346*) 

	Cons_Actionneur_Registre_Ext_m3h	: REAL;
	Cons_Actionneur_Registre_Souf_m3h 	: REAL;

(*Lecture de la temporisation du mode dépollution*)
	Lect_Temp_Seconde_Depol 			AT %MW7310: REAL; (*Adresse Modbus GTC : 19598*)
	Lect_Temp_Minute_Depol 				AT %MW7312: REAL; (*Adresse Modbus GTC : 19600*)
	Lect_Temp_heure_Depol 				AT %MW7314: REAL; (*Adresse Modbus GTC : 19602*)

(*Com RS485 Registre Soufflage*)
	Com_Ok_Reg_Souf 					: BOOL;
	Error_Com_Reg_Souf 					: BOOL;

	ValeursLues_Reg_Souf  				:ARRAY[1..4] OF INT;
	ValeursLues_Reg_Souf2  				:ARRAY[1..2] OF INT;
	ValeursLues_Reg_Souf3  				:ARRAY[1..2] OF INT;

	Posi_Relative_Reg_Souf 				: INT;
	Debit_Relative_Reg_Souf 			: INT;
	Lecture_Etat_Reg_Souf 				: INT;
	Lecture_ls_m3h_Reg_Souf 			: INT;
	Lecture_Software_Souf 				: INT;

	Posi_Absolue_Reg_Souf 		 		:INT;
	Debit_Absolue_Reg_Souf 				: INT;
	Lecture_Override_Control_Souf 		: INT;
	Lecture_Cons_Btw_Reg_Souf 			: INT;

	Lecture_Installation_Reg_Souf 		AT %MW9060: INT; (*Adresse Modbus GTC : 21348*)
	Lecture_Cons_Max_Reg_Souf 			AT %MW9061: INT; (*Adresse Modbus GTC : 21349*)
	Lecture_Cons_Min_Reg_Souf 			AT %MW9062: INT; (*Adresse Modbus GTC : 21350*)
	Lecture_Adresse_Reg_Souf 			AT %MW9063: INT; (*Adresse Modbus GTC : 21351*)
	Lecture_Self_Test_Reg_Souf 			AT %MW9064: INT; (*Adresse Modbus GTC : 21352*)


	Enable_ecr_param_Reg_Souf AT %MX17436.0:BOOL; (*Adresse Modbus GTC : 21006 bit 0*)

(*Com RS485 Registre Extraction*)
	Com_Ok_Reg_Extraction 				: BOOL;
	Error_RS485_Reg_Ext 				: BOOL;

	ValeursLues_Reg_Extraction  		 :ARRAY[1..4] OF INT;

	Posi_Relative_Reg_Extraction 		: INT;
	Debit_Relative_Reg_Extraction 		: INT;
	Posi_Absolue_Reg_Extraction 		: INT;
	Debit_Absolue_Reg_Extraction 		: INT;

	Ecriture_ls_m3h_Reg_Extraction 		: INT;
	Lecture_ls_m3h_Reg_Extraction 		: INT;
	Lecture_Override_Control_Ext 		: INT;
	Ecriture_Override_Control_Ext 		: INT;
	Lecture_Software_Ext 				: INT;
	Lecture_Etat_Reg_Extraction 		: INT;

(******************************************************************************************)
(*GESTION DES VARIABLES DE LA PARTIE ENCEINTE CLIMATIQUES*)
(******************************************************************************************)

(*Autres (Non utilisé dans la table d'échange)*)
	(*Gestion des états*)
	Mode_MEnCond						: BOOL;
	Mode_Fctnmt							: BOOL;
	Defaut_General_Humi 				:BOOL;
	Defaut_Arret_Mode25 				:BOOL;
	Dmd_Post_Ventilation				: BOOL;
	(*Autres*)
	RS_MEnCond: RS;
	(*Gestion des regulations*)
	(*Regule température*)
	Enable_Regul_PID_Temp 				:BOOL;
	Enable_Regul_PID_Temp_Chaud 		:BOOL;
	Enable_Regul_PID_Temp_Froid 		:BOOL;
	S_Cmd_Regul_PID_Temp_Chaud 			:REAL;
	S_Cmd_Regul_PID_Temp_Froid 			:REAL;
	(*Regule hygrométrie*)
	Enable_Regul_PID_Hr 				:BOOL;
	Enable_Regul_PID_Humi 				:BOOL;
	Enable_Regul_PID_Deshu 				:BOOL;
	S_Cmd_Regul_PID_Humi 				:REAL;
	S_Cmd_Regul_PID_Deshu 				:REAL;
	(*Gestion sortie d'ecart*)
	S_Ecart_Regul_PID_Temp 				:REAL;
	S_Ecart_Regul_PID_Hygro 			:REAL;
	(*Lecture des consignes appliquées*)
	Lect_Cons_Temperature_Cabine		: REAL;
	Lect_Cons_Hygrometrie_Cabine		: REAL;
	Lect_Cons_VitMot_Cabine_MEnCond		: REAL;
	MotRep_CTA						: Moteur_EC;
	MotSouf_CTA						: Moteur_EC;

(*Gestion des défauts*)
	Defaut_MotRep_CTA					:BOOL;
	Defaut_MotSouf_CTA					:BOOL;
	Defaut_Hygrostat_CTA 				:BOOL;
	Defaut_Alim_BatElec_CTA				:BOOL;
	Defaut_Humi_CTA						:BOOL;

	Defaut_Regul_Temp					:BOOL;
	Defaut_Regul_Hygro					:BOOL;
	Defaut_Discord_Souf_CTA				:BOOL;
	Defaut_Thermostat_Secu				:BOOL;

(*Lectures des consignes et des commandes Actionneurs*)
	Cons_Actionneur_V3V_Froid_CTA		AT %MW9066:REAL; (*Adresse Modbus GTC : 21354*)
	Cons_Actionneur_Mot1_Souf_CTA		AT %MW9068:REAL; (*Adresse Modbus GTC : 21356*)
	Cons_Actionneur_Mot2_Souf_CTA		AT %MW9070:REAL; (*Adresse Modbus GTC : 21358*)
	Cons_Actionneur_BatElec_CTA			AT %MW9072:REAL; (*Adresse Modbus GTC : 21360*)
	Cons_Actionneur_Humi_CTA			AT %MW9074:REAL; (*Adresse Modbus GTC : 21362*)

	Cmd_Actionneur_BatElec_CTA			:BOOL;
	Cmd_Actionneur_Humi_CTA				:BOOL;
END_VAR

(*===========================================================================*)
(*===========================================================================*)
(*===========================================================================*)
(*===========================================================================*)

VAR_GLOBAL PERSISTENT
(******************************************************************************************)
(*GESTION DES VARIABLES DE LA CABINE*)
(******************************************************************************************)

(*Consigne non récupérer sur la gtc et l'écran*)
	Own_Ip_Adress 						:STRING; 	(*Adresse Ip de l'automate à renseigner*)
	(*Variable PID*)
	Gain_PID_Bas_Deb_Ext				: REAL;
	Integral_PID_Bas_Deb_Ext			: REAL;
	Derivee_PID_Bas_Deb_Ext				: REAL;
	Gain_PID_Temp_Amb					: REAL;
	Integral_PID_Temp_Amb				: REAL;
	Derivee_PID_Temp_Amb				: REAL;
	Gain_PID_Press_Cab					: REAL;
	Integral_PID_Press_Cab				: REAL;
	Derivee_PID_Press_Cab				: REAL;
	Gain_PID_Temp_Eau_Mitig				: REAL;
	Integral_PID_Temp_Eau_Mitig			: REAL;
	Derivee_PID_Temp_Eau_Mitig			: REAL;
	(*Gestion des tolérance pour RAZ*)
	TOL_RAZ_MES_Deb_Souf 				:INT;
	TOL_RAZ_MES_Deb_Ext 				:INT;
	TOL_RAZ_MES_Petit_Deb 				:INT;
	TOL_RAZ_MES_Bypass 					:INT;
	TOL_Debit_Extraction 				:REAL;
	TOL_Debit_Soufflage 				:REAL;
	TOL_Deb_Ext_Reg_Ferm 				:REAL;
	TOL_Deb_Souf_Reg_Ferm 				:REAL;
	TOL_Regul_Press 					:REAL;
	(*Gestion ouverture de l'eau*)
	Cons_J_Forc_Vid_Lavabo 				:WORD;
	Cons_H_Forc_Vid_Lavabo 				:WORD;
	Cons_M_Forc_Vid_Lavabo 				:WORD;
	(*Couleur led mode libre*)
	Cde_Rouge_Cabine_Libre				:WORD;
	Cde_Vert_Cabine_Libre				:WORD;
	Cde_Bleu_Cabine_Libre				:WORD;
	Cde_Blanc_Cabine_Libre				:WORD;

	(* Paramètres registre ultrasson soufflage *)
	Ecriture_Installation_Reg_Souf 		AT %MW7992: INT; (*Adresse Modbus GTC : 20280*)
	Ecriture_Cons_Max_Reg_Souf 			AT %MW7993: INT; (*Adresse Modbus GTC : 20281*)
	Ecriture_Cons_Min_Reg_Souf 			AT %MW7994: INT; (*Adresse Modbus GTC : 20282*)
	Ecriture_Adresse_Reg_Souf 			AT %MW7995: INT; (*Adresse Modbus GTC : 20283*)
	Ecriture_Self_Test_Reg_Souf 		AT %MW7996: INT; (*Adresse Modbus GTC : 20284*)
	Ecriture_Cons_Btw_Reg_Souf 			: INT;
	Ecriture_Override_Control_Souf 		: INT;
	Ecriture_ls_m3h_Reg_Souf 			: INT; (*1=m3/h*)

(*Consigne non clasée*)
	Numero_Recette_Sel 					AT %MW7732: INT;  (*Adresse Modbus GTC : 20020*)
	Volume_Cabine						AT %MW7734: REAL; (*Adresse Modbus GTC : 20022*)
	Cons_Moteur_ByPass					AT %MW7736: REAL; (*Adresse Modbus GTC : 20024*)
	Cons_Temp_Amb						AT %MW7738: REAL; (*Adresse Modbus GTC : 20026*)
	Cons_Press_Cab						AT %MW7976: REAL; (*Adresse Modbus GTC : 20264*)
	Cons_Temp_EauMitige					AT %MW7998: REAL; (*Adresse Modbus GTC : 20286*)

(*Gestion des différents Tableau*)
	Tab_Nom_Recette						AT %MW141: ARRAY [1..2, 0..20] OF STRING(39); (*Adresse Modbus GTC : 12429*)
	Tab_Nom_Mode						AT %MW981: ARRAY [1..2, 1..30] OF STRING(31); (*Adresse Modbus GTC : 13269*)
	Tab_Mode_Texte						AT %MW1941: ARRAY [1..2, 30..60] OF STRING(139); (*Adresse Modbus GTC : 14229*)
	Tab_Enr_Recette						AT %MW6302: ARRAY[0..0, 1..30, 1..15] OF REAL; (*Adresse Modbus GTC : 18590*)
	Tab_Recette_Auto					: ARRAY[0..20, 1..30, 1..15] OF REAL;
	Tab_Enr_Mode_Manu					: ARRAY[1..15] OF REAL;

(* gestion Horodatage *)
	RTC_Modifiable						: TIMESTRUCT;
	rtcTime								: TIMESTRUCT;
	rtcMicro							: DWORD;
	Ecr_Annee_Automate					: WORD;
	Ecr_Mois_Automate					: WORD;
	Ecr_Jour_Automate					: WORD;
	Ecr_Heure_Automate					: WORD;
	Ecr_Minute_Automate					: WORD;

	deb_lundi							AT %MW7711: INT; (*Adresse Modbus GTC : 19999*)
	Fin_Lundi							AT %MW7712: INT; (*Adresse Modbus GTC : 20000*)
	deb_Mardi							AT %MW7713: INT; (*Adresse Modbus GTC : 20001*)
	Fin_Mardi							AT %MW7714: INT; (*Adresse Modbus GTC : 20002*)
	deb_Mercredi						AT %MW7715: INT; (*Adresse Modbus GTC : 20003*)
	Fin_Mercredi						AT %MW7716: INT; (*Adresse Modbus GTC : 20004*)
	deb_Jeudi							AT %MW7717: INT; (*Adresse Modbus GTC : 20005*)
	Fin_Jeudi							AT %MW7718: INT; (*Adresse Modbus GTC : 20006*)
	deb_Vendredi						AT %MW7719: INT; (*Adresse Modbus GTC : 20007*)
	Fin_Vendredi						AT %MW7720: INT; (*Adresse Modbus GTC : 20008*)
	deb_Samedi							AT %MW7721: INT; (*Adresse Modbus GTC : 20009*)
	Fin_Samedi							AT %MW7722: INT; (*Adresse Modbus GTC : 20010*)
	deb_Dimanche						AT %MW7723: INT; (*Adresse Modbus GTC : 20011*)
	Fin_Dimanche						AT %MW7724: INT; (*Adresse Modbus GTC : 20012*)

(*Gestion des forçages*)
	F_Cons_Registre_Extraction 			AT %MW7725: INT; (*Adresse Modbus GTC : 20013*)
	F_Cons_Registre_Soufflage 			AT %MW7726: INT; (*Adresse Modbus GTC : 20014*)
	F_Cons_Reg_Etanche_Ext				AT %MW7974: REAL; (*Adresse Modbus GTC : 20262*)
	F_Cons_V3V_Eau_Mitig				AT %MW7978: REAL; (*Adresse Modbus GTC : 20266*)

(* Gestion des consignes de la lumière *)
	Cons_Dimmer_Auto					AT %MW7727: INT; (*Adresse Modbus GTC : 20015*)
	Cons_Appl_Rouge_Auto				AT %MW7728: INT; (*Adresse Modbus GTC : 20016*)
	Cons_Appl_Vert_Auto					AT %MW7729: INT; (*Adresse Modbus GTC : 20017*)
	Cons_Appl_Bleu_Auto					AT %MW7730: INT; (*Adresse Modbus GTC : 20018*)
	Cons_Appl_Blanc_Auto				AT %MW7731: INT; (*Adresse Modbus GTC : 20019*)

(*Gestion du trop plein*)
	Garde_Deau_Douche 					AT %MW7740: REAL; (*Adresse Modbus GTC : 20028*)
	Garde_Deau_Lavabo 					AT %MW7742: REAL; (*Adresse Modbus GTC : 20030*)
	Trop_Plein_Douche 					AT %MW7744: REAL; (*Adresse Modbus GTC : 20032*)
	Trop_Plein_Lavabo 					AT %MW7746: REAL; (*Adresse Modbus GTC : 20034*)
	Coef_Correction_DebitEau			: REAL;

(*Consigne mode manu*)
	Manu_Choix_Numero_Mode 				AT %MW7748: REAL; (*Adresse Modbus GTC : 20036*)
	Manu_Tempo_Transition_Seconde		AT %MW7750: REAL; (*Adresse Modbus GTC : 20038*)
	Manu_Tempo_Transition_Minute 		AT %MW7752: REAL; (*Adresse Modbus GTC : 20040*)
	Manu_Tempo_Transition_Heure 		AT %MW7754: REAL; (*Adresse Modbus GTC : 20042*)
	Manu_Lct_Cons_Vol_Douche			AT %MW7756: REAL; (*Adresse Modbus GTC : 20044*)
	Manu_Lct_Cons_Vol_Lavabo			AT %MW7758: REAL; (*Adresse Modbus GTC : 20046*)
	Manu_Cons_Deb_Soufflage				AT %MW7760: REAL; (*Adresse Modbus GTC : 20048*)
	Manu_Cons_Deb_Extraction			AT %MW7762: REAL; (*Adresse Modbus GTC : 20050*)
	Manu_Cons_Temp_Eau					AT %MW7764: REAL; (*Adresse Modbus GTC : 20052*)
	Manu_Cons_Nbre_Chasse				AT %MW7766: REAL; (*Adresse Modbus GTC : 20054*)
	Manu_Cons_Para11					AT %MW7768: REAL; (*Adresse Modbus GTC : 20056*)
	Manu_Cons_Para12					AT %MW7770: REAL; (*Adresse Modbus GTC : 20058*)
	Manu_Cons_Para13					AT %MW7772: REAL; (*Adresse Modbus GTC : 20060*)
	Manu_Cons_Para14 					AT %MW7774: REAL; (*Adresse Modbus GTC : 20062*)
	Manu_Cons_Para15 					AT %MW7776: REAL; (*Adresse Modbus GTC : 20064*)

(*Temporisation de sécurisation des alimentations*)
	Temp_Secu_Debord_Douche				AT %MW7778: INT; (*Adresse Modbus GTC : 20066*)
	Temp_Secu_Debord_Lavabo				AT %MW7780: INT; (*Adresse Modbus GTC : 20068*)
	Volume_Secu_Debord_Douche			AT %MW9810:INT; (*Adresse Modbus GTC : 22098*)
	Volume_Secu_Debord_Lavabo			AT %MW9812:INT; (*Adresse Modbus GTC : 22100*)
	Temps_Remplissage_WC				:INT;

(*Gestion des consignes de regulation d'air*)
	Cons_Deb_Souf_Etat_Libre			AT %MW7782: REAL; (*Adresse Modbus GTC : 20070*)
	Cons_Deb_Ext_Etat_Libre				AT %MW7784: REAL; (*Adresse Modbus GTC : 20072*)

	Cons_Deb_Souf_Etat_Depol			AT %MW7786: REAL; (*Adresse Modbus GTC : 20074*)
	Cons_Deb_PD_Etat_Depol				AT %MW7788: REAL; (*Adresse Modbus GTC : 20076*)

	Cons_Deb_Souf_Mode_Focnt	 		AT %MW7790: REAL; (*Adresse Modbus GTC : 20078*)
	Cons_Deb_Ext_Mode_Focnt				AT %MW7792: REAL; (*Adresse Modbus GTC : 20080*)

	Cons_Deb_Souf_Mode_MEC				AT %MW7794: REAL; (*Adresse Modbus GTC : 20082*)
	Cons_Deb_Ext_Mode_MEC				AT %MW7796: REAL; (*Adresse Modbus GTC : 20084*)
	
	Cons_Deb_Souf_Etat_Nettoyage 		: REAL;
	Cons_Deb_Ext_Etat_Nettoyage			: REAL;

	Cons_Deb_Souf_Etat_Evaluation 		: REAL;
	Cons_Deb_Ext_Etat_Evaluation		: REAL;

(*	
	Cons_Deb_Souf_Etat_Nettoyage 		AT %MW7790: REAL; (*Adresse Modbus GTC : 20078*)
	Cons_Deb_Ext_Etat_Nettoyage			AT %MW7792: REAL; (*Adresse Modbus GTC : 20080*)

	Cons_Deb_Souf_Etat_Evaluation 		AT %MW7794: REAL; (*Adresse Modbus GTC : 20082*)
	Cons_Deb_Ext_Etat_Evaluation		AT %MW7796: REAL; (*Adresse Modbus GTC : 20084*)
*)

	Cons_Max_Bas_Deb_Ext				AT %MW7798: REAL; (*Adresse Modbus GTC : 20086*)
	Cons_Min_Bas_Deb_Ext				AT %MW7800: REAL; (*Adresse Modbus GTC : 20088*)

(*Gestion des consignes de temporisation de la dépollution*)
	Cons_Temp_Minute_Depol 				AT %MW7802: REAL; (*Adresse Modbus GTC : 20090*)
	Cons_Temp_heure_Depol 				AT %MW7804: REAL; (*Adresse Modbus GTC : 20092*)

(*Gestion des objets actionenurs*)
	Tab_Mot_Aerobox_Bas_Deb				AT %MW7806:Objet_Moteur_EC; (*Adresse Modbus GTC : 20094*)
	Tab_Batterie_Elec					AT %MW7826:Objet_BatElec; (*Adresse Modbus GTC : 20114*)
	Tab_Mot_ByPass						AT %MW7846:Objet_Moteur_EC; (*Adresse Modbus GTC : 20134*)

(*Gestion des objets sondes*)
	Tab_MES_Sonde_Temp_Amb 				AT %MW7866:Objet_Sonde; (*Adresse Modbus GTC : 20154*)
	Tab_MES_Sonde_Hygro_Amb 			AT %MW7878:Objet_Sonde; (*Adresse Modbus GTC : 20166*)
	Tab_MES_Sonde_Gros_Debit_Soufflage 	AT %MW7890:Objet_Sonde; (*Adresse Modbus GTC : 20178*)
	Tab_MES_Sonde_Gros_Debit_Extraction AT %MW7902:Objet_Sonde; (*Adresse Modbus GTC : 20190*)
	Tab_MES_Sonde_Petit_Debit_Extraction AT %MW7914:Objet_Sonde; (*Adresse Modbus GTC : 20202*)
	Tab_MES_Sonde_Debit_Alim_Douche 	AT %MW7926:Objet_Sonde; (*Adresse Modbus GTC : 20214*)
	Tab_MES_Sonde_Debit_Alim_Lavabo 	AT %MW7938:Objet_Sonde; (*Adresse Modbus GTC : 20226*)
	Tab_MES_Sonde_Press_Cab				AT %MW7950:Objet_Sonde; (*Adresse Modbus GTC : 20238*)
	Tab_MES_Sonde_Press_ByPass 			AT %MW7962:Objet_Sonde; (*Adresse Modbus GTC : 20250*)
	Tab_MES_Sonde_Temp_Eau_Mitig 		AT %MW7980:Objet_Sonde; (*Adresse Modbus GTC : 20268*)

	Tab_Mes_Sonde_Temp_BatEG			AT %MW9746:Objet_Sonde; (*Adresse Modbus GTC : 22034*)
	Tab_Mes_Sonde_Pression_Souf			AT %MW9786:Objet_Sonde; (*Adresse Modbus GTC : 22074*)
	Tab_Mes_Sonde_Pression_Ext			AT %MW9798:Objet_Sonde; (*Adresse Modbus GTC : 22086*)
	Tab_Mes_Sonde_Temp_Souf				AT %MW8238:Objet_Sonde; (*Adresse Modbus GTC : 20526*)

(* Gestion des ecritures et lectures des bits *)
	//Ecr_Bit_Cmd_IHM1 AT %MW17422: INT; (*Adresse Modbus GTC : 20999*)
	//Ecr_Bit_Cmd_IHM2 AT %MW17424: INT; (*Adresse Modbus GTC : 21000*)
	//Ecr_Bit_Cmd_IHM3 AT %MW17426: INT; (*Adresse Modbus GTC : 21001*)
	//Ecr_Bit_Cmd_IHM4 AT %MW17428: INT; (*Adresse Modbus GTC : 21002*)
	//Ecr_Bit_Cmd_IHM5 AT %MW17430: INT; (*Adresse Modbus GTC : 21003*)
	//Ecr_Bit_Cmd_IHM6 AT %MW17432: INT; (*Adresse Modbus GTC : 21004*)
	//Ecr_Bit_Cmd_IHM7 AT %MW17434: INT; (*Adresse Modbus GTC : 21005*)
	//Ecr_Bit_Cmd_IHM8 AT %MW17436: INT; (*Adresse Modbus GTC : 21006*)
	//Ecr_Bit_Cmd_IHM9 AT %MW17438: INT; (*Adresse Modbus GTC : 21007*)
	//Ecr_Bit_Cmd_IHM10 AT %MW17440: INT; (*Adresse Modbus GTC : 21008*)

	//Lect_Bit_IHM1 AT %MW17442: INT; (*Adresse Modbus GTC : 21009*)
	//Lect_Bit_IHM2 AT %MW17444: INT; (*Adresse Modbus GTC : 21010*)
	//Lect_Bit_IHM3 AT %MW17446: INT; (*Adresse Modbus GTC : 21011*)
	//Lect_Bit_IHM4 AT %MW17448: INT; (*Adresse Modbus GTC : 21012*)
	//Lect_Bit_IHM5 AT %MW17450: INT; (*Adresse Modbus GTC : 21013*)
	//Lect_Bit_IHM6 AT %MW17452: INT; (*Adresse Modbus GTC : 21014*)
	//Lect_Bit_IHM7 AT %MW17454: INT; (*Adresse Modbus GTC : 21015*)
	//Lect_Bit_IHM8 AT %MW17456: INT; (*Adresse Modbus GTC : 21016*)
	//Lect_Bit_IHM9 AT %MW17458: INT; (*Adresse Modbus GTC : 21017*)
	//Lect_Bit_IHM10 AT %MW17460: INT; (*Adresse Modbus GTC : 21018*)	

(*Bit ecriture gestion recette*)
	Start_Mode_Manu						AT %MX17422.0: BOOL; (*Adresse Modbus GTC : 20999 bit 0*)
	Reset_Mode_Manu						AT %MX17422.1: BOOL; (*Adresse Modbus GTC : 20999 bit 1*)
	Start_Etat_Depollution				AT %MX17422.2: BOOL; (*Adresse Modbus GTC : 20999 bit 2*)
	Start_Etat_Nettoyage				AT %MX17422.3: BOOL; (*Adresse Modbus GTC : 20999 bit 3*)
	Activation_Ecl						AT %MX17422.4: BOOL; (*Adresse Modbus GTC : 20999 bit 4*)
	Choix_Langue						AT %MX17422.5: BOOL; (*Adresse Modbus GTC : 20999 bit 5*) (*0=Français / 1=Américain*)
	Valid_Texte							AT %MX17422.6: BOOL; (*Adresse Modbus GTC : 20999 bit 6*)
	Bp_Pause							AT %MX17422.7: BOOL; (*Adresse Modbus GTC : 20999 bit 7*)
	Detail_Nom_Recette_Mode				AT %MX17422.8: BOOL; (*Adresse Modbus GTC : 20999 bit 8*)
	Validation_Recette_Auto				AT %MX17422.9: BOOL; (*Adresse Modbus GTC : 20999 bit 9*)
	Start_Recette_Mode_Auto				AT %MX17422.10: BOOL;(*Adresse Modbus GTC : 20999 bit 10*)
	Reset_Mode_Auto						AT %MX17422.11: BOOL; (*Adresse Modbus GTC : 20999 bit 11*)
	Cmd_Rearmement						AT %MX17422.12: BOOL; (*Adresse Modbus GTC : 20999 bit 12*)
	Cmd_Enr_Recette						AT %MX17422.13: BOOL; (*Adresse Modbus GTC : 20999 bit 13*)
	Cmd_Mode_Maintenance				AT %MX17422.14: BOOL; (*Adresse Modbus GTC : 20999 bit 14*)	
	
(*Gestion des options*)
	(*Option types de cabine*)
	Option_Cabine_Seche 				AT %MX17426.0: BOOL; (*Adresse Modbus GTC : 21001 bit 0*)
	Option_Cabine_Humide 				AT %MX17426.1: BOOL; (*Adresse Modbus GTC : 21001 bit 1*)
	Option_Cabine_Climatique 			AT %MX17428.15: BOOL; (*Adresse Modbus GTC : 21002 bit 15*)

	(*Option actionneurs*)
	Option_Douche						AT %MX17426.2: BOOL; (*Adresse Modbus GTC : 21001 bit 2*)
	Option_Lavabo 						AT %MX17426.3: BOOL; (*Adresse Modbus GTC : 21001 bit 3*)
	Option_Douchette 					AT %MX17426.4: BOOL; (*Adresse Modbus GTC : 21001 bit 4*)
	Option_NEP							AT %MX17428.14: BOOL; (*Adresse Modbus GTC : 21002 bit 14*)
	Option_Prise 						AT %MX17426.5: BOOL; (*Adresse Modbus GTC : 21001 bit 5*)
	Option_WC_GV 						AT %MX17424.0: BOOL; (*Adresse Modbus GTC : 21000 bit 0*)
	Option_WC_PV 						AT %MX17424.1: BOOL; (*Adresse Modbus GTC : 21000 bit 1*)
	Option_RegSouf_Ultrason 			AT %MX17428.12: BOOL; (*Adresse Modbus GTC : 21002 bit 12*)
	Option_Reg_Etanche_Ext 				AT %MX17428.8: BOOL; (*Adresse Modbus GTC : 21002 bit 0*)
	Option_V3V_EauMitig 				AT %MX17426.8: BOOL; (*Adresse Modbus GTC : 21001 bit 8*)
	Option_RegExt_Ultrason 				AT %MX17428.13: BOOL; (*Adresse Modbus GTC : 21002 bit 13*)
	Option_Reg_Etanche_Souf 			AT %MX17428.7: BOOL; (*Adresse Modbus GTC : 21002 bit 7*)
	Option_Bas_Debit					AT %MX17426.10: BOOL; (*Adresse Modbus GTC : 21001 bit 10*)
	Option_Batt_Elec 					AT %MX17428.3: BOOL; (*Adresse Modbus GTC : 21002 bit 3*)
	Option_Mot_ByPass 					AT %MX17428.4: BOOL; (*Adresse Modbus GTC : 21002 bit 4*)
	Option_Pompe_De_Relevage 			AT %MX17426.13: BOOL; (*Adresse Modbus GTC : 21001 bit 13*)

	(*Option capteurs*)
	Option_Debitmetre_Douche 			AT %MX17428.1: BOOL; (*Adresse Modbus GTC : 21002 bit 1*)
	Option_Debitmetre_Lavabo 			AT %MX17428.2: BOOL; (*Adresse Modbus GTC : 21002 bit 2*)
	Option_Sonde_Temp_Hygro_Amb 		AT %MX17426.11: BOOL; (*Adresse Modbus GTC : 21001 bit 11*)
	Option_Capteur_Press_Cab 			AT %MX17428.6: BOOL; (*Adresse Modbus GTC : 21002 bit 6*)
	Option_Press_SoufExt_General 		AT %MX17426.7: BOOL; (*Adresse Modbus GTC : 21001 bit 7*)
	Option_Sonde_Temp_EauMitig 			AT %MX17424.2: BOOL; (*Adresse Modbus GTC : 21000 bit 2*)
	Option_Temp_Batterie_EG 			AT %MX17424.3: BOOL; (*Adresse Modbus GTC : 21000 bit 3*)
	Option_Sonde_Temp_Amb 				AT %MX17426.12: BOOL; (*Adresse Modbus GTC : 21001 bit 12*)
	Option_Contact_Porte 				AT %MX17428.0: BOOL; (*Adresse Modbus GTC : 21002 bit 0*)
	Option_Niveau_Haut_Douche 			AT %MX17426.14: BOOL; (*Adresse Modbus GTC : 21001 bit 14*)
	Option_Niveau_Haut_Lavabo 			AT %MX17426.15: BOOL; (*Adresse Modbus GTC : 21001 bit 15*)
	Option_Defaut_Prise_Elec 			AT %MX17428.10: BOOL; (*Adresse Modbus GTC : 21002 bit 10*)

	(*Option communication*)
	Option_InterCom 					AT %MX17426.6: BOOL; (*Adresse Modbus GTC : 21001 bit 6*)
	Option_Com_RegSouf_Ultrason			AT %MX17428.5: BOOL; (*Adresse Modbus GTC : 21002 bit 5*)
	Option_Com_RegExt_Ultrason 			AT %MX17428.11: BOOL; (*Adresse Modbus GTC : 21002 bit 0*)

	(*Option régulations*)
	Option_Regul_Deb_Ou_Press 			AT %MX17428.9: BOOL; (*Adresse Modbus GTC : 21002 bit 8*)(*0=Deb 1=press*)
	Option_Regul_Temp_Eau				AT %MX17426.9: BOOL; (*Adresse Modbus GTC : 21001 bit 9*)

(*Gestion des forçages*)
	EF_Cmd_PC_Cab  						AT %MX17430.0: BOOL;
	EF_Cmd_Vanne_Alim_Douche  			AT %MX17430.1: BOOL;
	EF_Cmd_Vanne_Alim_Douchette  		AT %MX17430.2: BOOL;
	EF_Cmd_Vanne_Alim_Lavabo  			AT %MX17430.3: BOOL;
	EF_Cmd_Vanne_Vid_Douche  			AT %MX17430.4: BOOL;
	EF_Cmd_Vanne_Vid_Lavabo 			AT %MX17430.5: BOOL;
	EF_Cmd_ElectroValve_Alim_Douche  	AT %MX17430.6: BOOL;
	EF_Cmd_ElectroValve_Alim_Lavabo 	AT %MX17430.7: BOOL;
	EF_Cons_Registre_Extraction 		AT %MX17430.8: BOOL;
	EF_Cons_Registre_Soufflage 			AT %MX17430.9: BOOL;
	EF_Vanne_Souf_Bas_Deb 				AT %MX17430.10: BOOL;
	EF_Vanne_Ext_Bas_Deb 				AT %MX17430.11: BOOL;
	EF_Cons_Reg_Etanche_Ext 			AT %MX17430.12: BOOL;
	EF_Cmd_Reg_Etanche_Souf 			AT %MX17430.13: BOOL;
	EF_Cons_V3V_Eau_Mitig 				AT %MX17430.14: BOOL;
	EF_Vanne_Alim_NEP 					AT %MX17430.15: BOOL;
	EF_Cons_V3V_Bat_Froid_CTA  			AT %MX17438.0: BOOL;
	EF_Cmd_Verin_WC_GV  				AT %MX17438.1: BOOL;
	EF_Cmd_Verin_WC_PV  				AT %MX17438.3: BOOL;

	F_Cmd_PC_Cab  						AT %MX17432.0: BOOL;
	F_Cmd_Vanne_Alim_Douche  			AT %MX17432.1: BOOL;
	F_Cmd_Vanne_Alim_Douchette  		AT %MX17432.2: BOOL;
	F_Cmd_Vanne_Alim_Lavabo  			AT %MX17432.3: BOOL;
	F_Cmd_Vanne_Vid_Douche  			AT %MX17432.4: BOOL;
	F_Cmd_Vanne_Vid_Lavabo 				AT %MX17432.5: BOOL;
	F_Cmd_ElectroValve_Alim_Douche  	AT %MX17432.6: BOOL;
	F_Cmd_ElectroValve_Alim_Lavabo 		AT %MX17432.7: BOOL;
	F_Vanne_Souf_Bas_Deb 				AT %MX17432.8: BOOL;
	F_Vanne_Ext_Bas_Deb 				AT %MX17432.9: BOOL;
	F_Cmd_Reg_Etanche_Souf 				AT %MX17432.10: BOOL;
	F_Vanne_Alim_NEP 					AT %MX17432.11: BOOL;
	F_Cmd_Verin_WC_GV  					AT %MX17438.2: BOOL; (*Impultion*)
	F_Cmd_Verin_WC_PV  					AT %MX17438.4: BOOL; (*Impultion*)

(*Bit horodatage*)
	Sel_Lundi  							AT %MX17434.0: BOOL;
	Sel_Mardi  							AT %MX17434.1: BOOL;
	Sel_Mercredi  						AT %MX17434.2: BOOL;
	Sel_Jeudi  							AT %MX17434.3: BOOL;
	Sel_Vendredi  						AT %MX17434.4: BOOL;
	Sel_Samedi 							AT %MX17434.5: BOOL;
	Sel_Dimanche  						AT %MX17434.6: BOOL;
	StartMiseALheure   					AT %MX17434.7: BOOL; (*Impultion*)
	
(******************************************************************************************)
(*GESTION DES VARIABLES DE LA PARTIE ENCEINTE CLIMATIQUES*)
(******************************************************************************************)
(*Consigne non récupérer sur la gtc et l'écran*)
	(*Gestion des tolérance pour RAZ*)
	TOL_Regul_Temp_EnceintClim 			:REAL;
	TOL_Regul_Hygro_EnceintClim 		:REAL;
	(*Gestion des regulations*)
	(*Regule température*)
	Offset_Regul_PID_Temp 				:REAL;
	Gain_Regul_PID_Temp_Chaud 			:REAL;
	Integral_Regul_PID_Temp_Chaud 		:REAL;
	Derive_Regul_PID_Temp_Chaud 		:REAL;
	Gain_Regul_PID_Souf_Chaud 			:REAL;
	Integral_Regul_PID_Souf_Chaud 		:REAL;
	Derive_Regul_PID_Souf_Chaud 		:REAL;
	Gain_Regul_PID_Temp_Froid 			:REAL;
	Integral_Regul_PID_Temp_Froid 		:REAL;
	Derive_Regul_PID_Temp_Froid 		:REAL;
	Limit_Max_Souf						:REAL;
	Limit_Min_Souf						:REAL;
	Kp_Ambiance							:REAL;
	Ki_Ambiance							:REAL;
	Kd_Ambiance							:REAL;
	(*Regule hygrométrie*)
	Offset_Regul_PID_Hr 				:REAL;
	Gain_Regul_PID_Humi 				:REAL;
	Integral_Regul_PID_Humi 			:REAL;
	Derive_Regul_PID_Humi 				:REAL;
	Gain_Regul_PID_Deshu 				:REAL;
	Integral_Regul_PID_Deshu 			:REAL;
	Derive_Regul_PID_Deshu 				:REAL;
	(*Gestion Mini Maxi des actionneurs*)
	Cons_Mini_V3V_Bat_Froid				:REAL;
	Cons_Maxi_V3V_Bat_Froid				:REAL;
	Cons_Maxi_Bat_Electrique 			:REAL;
	Cons_Maxi_Humidificateur 			:REAL;
	Cons_Maxi_Mot1_CTA	 				:REAL;
	Cons_Maxi_Mot2_CTA	 				:REAL;
	(*A classer*)
	Cons_Sec_Post_Ventil				:INT;
	Mini_Decal_PID_Deshu				:REAL;
	Maxi_Decal_PID_Deshu				:REAL;
	Mini_Decal_Deshu					:REAL;
	Maxi_Decal_Deshu					:REAL;

(*Gestion des consignes de fonctionnement de l'enceinte climatique*)
	Cons_Temperature_Cabine				AT %MW8000: REAL; (*Adresse Modbus GTC : 20288*)
	Cons_Hygrometrie_Cabine				AT %MW8002: REAL; (*Adresse Modbus GTC : 20290*)
	Cons_VitMot_Cabine_MEnCond			AT %MW8004: REAL; (*Adresse Modbus GTC : 20292*)
	Cons_VitMot_Cabine_EnCond			AT %MW8006: REAL; (*Adresse Modbus GTC : 20294*)

(*Gestion des Objets*)
	Tab_MotRep_CTA						AT %MW8010: Objet_Moteur_EC; (*Adresse Modbus GTC : 20298*)
	Tab_MotSouf_CTA						AT %MW8030: Objet_Moteur_EC; (*Adresse Modbus GTC : 20318*)
	Tab_Batterie_Elec_CTA				AT %MW8050: Objet_BatElec; (*Adresse Modbus GTC : 20338*)

(*Gestion des forçages*)
	F_Cons_V3V_Bat_Froid_CTA 			AT %MW8008:REAL; (*Adresse Modbus GTC : 20296*)
END_VAR

// ---- Global Variables/GVL_RegTROX.TcGVL
{attribute 'qualified_only'}
VAR_GLOBAL PERSISTENT
	//Déclaration des tables de structure des sondes
	TAB_Sonde_RegSouf_GD_FCVT01			AT %MW8070:Objet_Sonde;
	TAB_Sonde_RegSouf_PD_FCVT02			AT %MW8082:Objet_Sonde;
	TAB_Sonde_RegSouf_Cabine_FCVT03		AT %MW8094:Objet_Sonde;
	TAB_Sonde_RegBypass_FCVT04			AT %MW8106:Objet_Sonde;
	TAB_Sonde_RegSouf_CabGD_FCVT05		AT %MW8118:Objet_Sonde;
	TAB_Sonde_RegSouf_CabPD_FCVT06		AT %MW8130:Objet_Sonde;
	TAB_Sonde_RegRep_FCVT07				AT %MW8142:Objet_Sonde;
	
	//Déclaration des tables de structure des registres
	TAB_Reg_RegSouf_GD_FCVT01			AT %MW8154:Objet_Registre;
	TAB_Reg_RegSouf_PD_FCVT02			AT %MW8166:Objet_Registre;
	TAB_Reg_RegSouf_Cabine_FCVT03		AT %MW8178:Objet_Registre;
	TAB_Reg_RegBypass_FCVT04			AT %MW8190:Objet_Registre;
	TAB_Reg_RegSouf_CabGD_FCVT05		AT %MW8202:Objet_Registre;	
	TAB_Reg_RegSouf_CabPD_FCVT06		AT %MW8214:Objet_Registre;
	TAB_Reg_RegRep_FCVT07				AT %MW8226:Objet_Registre;

	//Consigne ades seuils de débit des registres
	ConsMax_FCVT01						AT %MW9092:REAL;
	ConsMin_FCVT01						AT %MW9094:REAL;
	
	ConsMax_FCVT02						AT %MW9096:REAL;
	ConsMin_FCVT02						AT %MW9098:REAL;
	
	ConsMax_FCVT03						AT %MW9100:REAL;
	ConsMin_FCVT03						AT %MW9102:REAL;
	
	ConsMax_FCVT04						AT %MW9104:REAL;
	ConsMin_FCVT04						AT %MW9106:REAL;
	
	ConsMax_FCVT05						AT %MW9108:REAL;
	ConsMin_FCVT05						AT %MW9110:REAL;
	
	ConsMax_FCVT06						AT %MW9112:REAL;
	ConsMin_FCVT06						AT %MW9114:REAL;
	
	ConsMax_FCVT07						AT %MW9116:REAL;
	ConsMin_FCVT07						AT %MW9118:REAL;
END_VAR

VAR_GLOBAL	
	//Déclaration des objets de mesure de débit
	MES_RegSouf_GD_FCVT01				:Objet_Sonde_V1;
	MES_RegSouf_PD_FCVT02				:Objet_Sonde_V1;
	MES_RegSouf_Cabine_FCVT03			:Objet_Sonde_V1;
	MES_RegBypass_FCVT04				:Objet_Sonde_V1;
	MES_RegSouf_CabGD_FCVT05			:Objet_Sonde_V1;
	MES_RegSouf_CabPD_FCVT06			:Objet_Sonde_V1;
	MES_RegRep_FCVT07					:Objet_Sonde_V1;
	
	//Déclaration des objets des registres
	RegSouf_GD_FCVT01					:Objet_Registre_V1;
	RegSouf_PD_FCVT02					:Objet_Registre_V1;
	RegSouf_Cabine_FCVT03				:Objet_Registre_V1;
	RegBypass_FCVT04					:Objet_Registre_V1;
	RegSouf_CabGD_FCVT05				:Objet_Registre_V1;
	RegSouf_CabPD_FCVT06				:Objet_Registre_V1;
	RegRep_FCVT07						:Objet_Registre_V1;
	
	//Déclaration des objets de la communication des registres
	Com_RegSouf_GD_FCVT01				:Com485_RegTROX;
	Com_RegSouf_PD_FCVT02				:Com485_RegTROX;
	Com_RegSouf_Cabine_FCVT03			:Com485_RegTROX;
	Com_Reg_Bypass_FCVT04				:Com485_RegTROX;
	Com_RegSouf_CabGD_FCVT05			:Com485_RegTROX;
	Com_RegSouf_CabPD_FCVT06			:Com485_RegTROX;
	Com_RegRep_FCVT07					:Com485_RegTROX;
	
	//Consigne appliquée de débit sur les registres
	ConsAppliDeb_RegSouf_GD_FCVT01		AT %MW9078:REAL;
	ConsAppliDeb_RegSouf_PD_FCVT02		AT %MW9080:REAL;
	ConsAppliDeb_RegSouf_Cabine_FCVT03	AT %MW9082:REAL;
	ConsAppliDeb_Reg_Bypass_FCVT04		AT %MW9084:REAL;
	ConsAppliDeb_RegSouf_CabGD_FCVT05	AT %MW9086:REAL;
	ConsAppliDeb_RegSouf_CabPD_FCVT06	AT %MW9088:REAL;
	ConsAppliDeb_RegRep_FCVT07			AT %MW9090:REAL;
	
	//Gestion des défauts
	RegSouf_GD_FCVT01_DefCom			:BOOL;
	RegSouf_GD_FCVT01_Def_DiscordDeb	:BOOL;
	
	RegSouf_PD_FCVT02_DefCom			:BOOL;
	RegSouf_PD_FCVT02_Def_DiscordDeb	:BOOL;
	
	RegSouf_Cabine_FCVT03_DefCom		:BOOL;
	RegSouf_Cabine_FCVT03_Def_DiscordDeb:BOOL;
	
	Reg_Bypass_FCVT04_DefCom			:BOOL;
	Reg_Bypass_FCVT04_Def_DiscordDeb	:BOOL;
	
	RegSouf_CabGD_FCVT05_DefCom			:BOOL;
	RegSouf_CabGD_FCVT05_Def_DiscordDeb	:BOOL;
	
	RegSouf_CabPD_FCVT06_DefCom			:BOOL;
	RegSouf_CabPD_FCVT06_Def_DiscordDeb	:BOOL;
	
	RegRep_FCVT07_DefCom				:BOOL;
	RegRep_FCVT07_Def_DiscordDeb		:BOOL;
END_VAR

// ---- Global Variables/GVL_Visu.TcGVL
{attribute 'qualified_only'}
VAR_GLOBAL
	//Les différents état et/ou information de l'écran
	Page_En_Cours 	:STRING;
	Connexion	 	:WSTRING;
	Etat_Connexion	:BOOL;
	Language	 	:STRING;
	
	//Gestion du mouvement des flèches dans la page dépollution
	Arrow_Up		:INT;
	Arrow_Down		:INT;
	
	//Etat pour l'objet moteur
	Etat_On			:BOOL;
	Etat_Off		:BOOL;
	Etat_Fault		:BOOL;
	
	On_Off_Anim		:BOOL;				//Variable qui me permet d'animé mes images
	On_Off_Anim_Rap	:BOOL;				//Variable qui me permet d'animé mes images en plus rapide
	On_Off_Anim_Lent:BOOL;				//Variable qui me permet d'animé mes images en plus lent
	Nom_Cabine_FR	:STRING;			//Variable qui stock le nom de la cabine en français
	Nom_Cabine_EN	:STRING;			//Variable qui stock le nom de la cabine en anglais
	
	//Variable de couleur de la cabine en fonction de son état
	Couleur_Cabine 	:DWORD;
	Couleur_Cabine2	: DWORD;
	
	//Gestion de la page Nettoyage
	Cmd_Img_Clean1	:BOOL;
	Cmd_Img_Clean2	:BOOL;
	Cmd_Img_Clean3	:BOOL;
	Cmd_Img_Clean4	:BOOL;
	Cmd_Img_Clean5	:BOOL;
	Cmd_Img_Clean6	:BOOL;
	Cmd_Img_Clean7	:BOOL;
	
	//Gestion de la page Sel_Recettes
	Visu_Btn_Start	:BOOL;
	
	//Gestion de la page Recet_EnCours	
	Visu_VolEau_Douche	:BOOL;
	Visu_VolEau_Lavabo	:BOOL;
	Visu_ChasseEau		:BOOL;
	Visu_Mes_Debit_Eau	:REAL;
	Visu_Debit_Eau		:BOOL;
	Visu_Tempo			:BOOL;
	
	//Gestion de la page Mode_Manu
	Visu_VolEau_Douche_Manu	:BOOL;
	Visu_VolEau_Lavabo_Manu	:BOOL;
	Visu_ChasseEau_Manu		:BOOL;
	Visu_Mes_Debit_Eau_Manu	:REAL;
	Visu_Debit_Eau_Manu		:BOOL;
	Manu_Choix_Numero_Mode_INT	:INT;
	Manu_i					:INT;
	Manu_j					:INT;
	Affich_Debit_Eau_Manu	:BOOL;
	Affich_Debit_Eau_Manu_Douche	:BOOL;
	Affich_Debit_Eau_Manu_Lavabo	:BOOL;
	Affich_ChasseEau_Manu	:BOOL;
	Visu_Temp_Manu			:BOOL;
	
	//gestion des alarmes
	Affichage_PopUp_HightLevel	:BOOL;
	Affichage_PopUp_Alarm		:BOOL;
END_VAR

VAR_GLOBAL PERSISTENT
	Numero_Cabine	:INT;					//Ecrire le numéro de la cabine
	Tab_Choix_Modes	:ARRAY[0..32] OF BOOL;	//Tableau de choix des modes
	Min_Mode_Manu	:INT;					//Paramétrer le numéro du premier mode à TRUE
	Max_Mode_Manu	:INT;					//Paramétrer le denrier mode à TRUE
END_VAR

// ---- Global Variables/Variable_Configuration.TcGVL
{attribute 'Tc2GvlVarNames'}
VAR_CONFIG
END_VAR

// ---- POUs/a1_MAIN.TcPOU
PROGRAM a1_MAIN
VAR
	FB_S_UPS_CX81xx :FB_S_UPS_CX81xx;
END_VAR

(******************Gestion UPS********************************)
FB_S_UPS_CX81xx(
	sNetID:='',
	iPLCPort:= 851,
	tTimeout:= DEFAULT_ADS_TIMEOUT,
	eUpsMode:= eSUPS_WrPersistData_Shutdown,
	ePersistentMode:= SPDM_2PASS);

(***********************Execution des taches***********************)
a2_Gestion_ES();
a3_Ecriture_Bit();
a4_Lecture_Bit();
a5_Ecriture_InterCom();
a6_Lecture_InterCom();
b_SCL_Mesures();
c_Gestion_Defaut();
d_Gestion_Pause_Modes();
e_Gestion_Horraire();
f_Gestion_Etats();
g_Gestion_Texte_Modes();
h_Enr_Recette();
i_Protocol_Auto();
j_Protocol_Manu();
l_Cons_LED();
n0_Regulation_Bas_Deb();
n1_Regulation_Press();
n2_Regulation_Temp();
n3_Regul_Temp_EauMitig();
o_Cons_Cmd_Actionneurs();
//p_Com_Modbus_RS485();
q_Gestion_Actionneurs_ANA();
r_Gestion_Actionneurs_TOR();
s_InterCom_Esclave();
t_Enr_Variables();
Visu();
Alarmes();
(***********************Execution des taches de la partie enceinte climatique***********************)
IF (Option_Cabine_Climatique)
	THEN
	B_Gestion_Defaut();
	C0_Gestion_Consignes();
	C_Regul_Temp();
	D_Regul_Humi();
	E_Cons_Cmd_Actionneurs();
	F_Gestion_Actionneurs();
	ELSE
	S_Cmd_BatElec_CTA			:= FALSE;
	S_Cmd_Humi_CTA				:= FALSE;
	S_Cons_V3V_Froid_CTA		:= 0;
	S_Cons_MotRep_CTA			:= 0;
	S_Cons_MotSouf_CTA			:= 0;
	S_Cons_BatElec_CTA			:= 0;
	S_Cons_Humi_CTA				:= 0;

	Defaut_MotRep_CTA			:= FALSE;
	Defaut_MotSouf_CTA			:= FALSE;
	Defaut_Hygrostat_CTA 		:= FALSE;
	Defaut_Alim_BatElec_CTA		:= FALSE;
	Defaut_Humi_CTA				:= FALSE;
	Defaut_Regul_Temp			:= FALSE;
	Defaut_Regul_Hygro			:= FALSE;
	Defaut_Arret_Mode25			:= FALSE;

	Cons_Actionneur_V3V_Froid_CTA	:= 0.0;
	Cons_Actionneur_Mot1_Souf_CTA	:= 0.0;
	Cons_Actionneur_Mot2_Souf_CTA	:= 0.0;
	Cons_Actionneur_BatElec_CTA		:= 0.0;
	Cons_Actionneur_Humi_CTA		:= 0.0;

	Cmd_Actionneur_BatElec_CTA		:= FALSE;
	Cmd_Actionneur_Humi_CTA		:= FALSE;
	Dmd_Post_Ventilation				:= FALSE;
END_IF;

END_PROGRAM

// ---- POUs/a2_Gestion_ES.TcPOU
PROGRAM a2_Gestion_ES
VAR
	Var_BOOL_Bidon :BOOL;
	Var_INT_Bidon :INT;
END_VAR

(**********************************************Configuration des Entrées*)
	E_Info_Niveau_Haut_Douche := 		Var_BOOL_Bidon;
	E_Info_Niveau_Haut_Lavabo := 		Var_BOOL_Bidon;
	E_Info_Contact_Porte := 			ETOR6_Info_Contact_Porte;
	E_Info_PC_Cab := 					ETOR3_Info_Ma_Prise;
	E_Etat_Evac_SaniDouche := 			Var_BOOL_Bidon;
	E_Info_Klixon_BattElec := 			Var_BOOL_Bidon;
	E_Defaut_Prise_Elec :=				Var_BOOL_Bidon;

	E_Vanne_Alim_Douche_Ouv := 			Var_BOOL_Bidon;
	E_Vanne_Alim_Douche_Ferm := 		Var_BOOL_Bidon;
	E_Vanne_Alim_Douchette_Ouv := 		Var_BOOL_Bidon;
	E_Vanne_Alim_Douchette_Ferm := 		Var_BOOL_Bidon;
	E_Vanne_Alim_Lavabo_Ouv := 			Var_BOOL_Bidon;
	E_Vanne_Alim_Lavabo_Ferm := 		Var_BOOL_Bidon;
	E_Vanne_Vidange_Douche_Ouv := 		Var_BOOL_Bidon;
	E_Vanne_Vidange_Douche_Ferm := 		Var_BOOL_Bidon;
	E_Vanne_Vidange_Lavabo_Ouv := 		ETOR1_Fdc_Va_Vid_Lavabo_Ouv;
	E_Vanne_Vidange_Lavabo_Ferm := 		ETOR2_Fdc_Va_Vid_Lavabo_Ferm;
	E_Vanne_Alim_NEP_Ouv := 			Var_BOOL_Bidon;
	E_Vanne_Alim_NEP_Ferm := 			Var_BOOL_Bidon;

	E_Vanne_Souf_Bas_Deb_Ouv :=			Var_BOOL_Bidon;
	E_Vanne_Souf_Bas_Deb_Ferm :=		Var_BOOL_Bidon;
	E_Vanne_Ext_Bas_Deb_Ouv :=			Var_BOOL_Bidon;
	E_Vanne_Ext_Bas_Deb_Ferm :=			Var_BOOL_Bidon;

	E_Sonde_Temp_Amb := 				EAN2_Sonde_Temp_Cabine;
	E_Sonde_Hygro_Amb := 				EAN3_Sonde_Hygro_Cabine;
	E_Sonde_Pression_Cabine :=			EAN5_Sonde_Pression_Cabine;
	E_Sonde_Temp_Eau_Mitig :=			Var_INT_Bidon;
	E_Sonde_press_Souf :=				EAN6_Sonde_press_Souf;
	E_Sonde_press_Ext :=				EAN8_Sonde_press_Ext;
	E_Sonde_Temp_Batt_EG :=				EAN4_Sonde_Temp_Batt_EG;

	E_Sonde_Gros_Debit_Soufflage := 	Var_INT_Bidon;
	E_Sonde_Gros_Debit_Extraction := 	Var_INT_Bidon;
	E_Sonde_Petit_Debit_Extraction := 	Var_INT_Bidon;
	E_Sonde_Pression_ByPass :=			Var_INT_Bidon;
	E_Retour_Pos_Reg_Etanche_Ext :=		EAN7_Retour_Pos_Reg_Etanche_Ext;

	E_Sonde_Debit_Alim_Douche :=		Var_INT_Bidon;
	E_Sonde_Debit_Alim_Lavabo := 		EAN1_Sonde_Debit_Eau_Lavabo;
	E_Sonde_Temp_Souf :=				EAN9_Sonde_Temp_Souf;

(**********************************************Configuration des Sorties*)
	STOR3_Cmd_Ma_Prise := 				S_Cmd_PC_Cab;
	Var_BOOL_Bidon := 					S_Cmd_Vanne_Alim_Douche;
	Var_BOOL_Bidon := 					S_Cmd_Vanne_Alim_Douchette;
	Var_BOOL_Bidon := 					S_Cmd_Vanne_Alim_Lavabo;
	Var_BOOL_Bidon := 					S_Cmd_Vanne_Vid_Douche;
	STOR2_Cmd_Va_Vid_Lavabo  := 		S_Cmd_Vanne_Vid_Lavabo;
	Var_BOOL_Bidon := 					S_Cmd_Vanne_NEP;
	Var_BOOL_Bidon :=					S_Cmd_Appli_Verin_WC_GV;
	Var_BOOL_Bidon :=					S_Cmd_Appli_Verin_WC_PV;

	Var_BOOL_Bidon := 					S_Cmd_ElectroValve_Alim_Douche;
	STOR1_Cmd_EV_Alim_Lavabo := 		S_Cmd_ElectroValve_Alim_Lavabo;

	Var_BOOL_Bidon := 					S_Cmd_BattElec;
	Var_BOOL_Bidon :=					S_Cmd_Vanne_Souf_Bas_Deb;
	Var_BOOL_Bidon :=					S_Cmd_Vanne_Ext_Bas_Deb;
	Var_BOOL_Bidon :=					S_Cmd_Reg_Etanche_Souf;

	Var_INT_Bidon :=				 	S_Cons_Registre_Extraction;
	Var_INT_Bidon := 					S_Cons_Registre_Soufflage;
	Var_INT_Bidon := 					S_Cons_Moteur_BasDebit;
	Var_INT_Bidon := 					S_Cons_Moteur_ByPass;
	Var_INT_Bidon := 					S_Cons_BattElec;
	SAN7_Cons_Ouv_Reg_Etanche_Ext :=	S_Cons_Reg_Etanche_Ext;
	Var_INT_Bidon :=					S_Cons_Ouv_V3V_Eau_Mitig;
	Var_INT_Bidon := 					S_Cons_Module_Sontay;

(*Configuration des Entrées et Sorties - Gestion des enceintes climatiques*)
	E_Def_MotRep_CTA := 				ETOR7_Def_MotRep_Souf_CTA;
	E_Def_MotSouf_CTA := 				ETOR8_Def_MotSouf_Souf_CTA;
	E_Hygrostat_Souf_CTA := 			ETOR10_Hygrostat_Souf_CT;
	E_Def_Alim_BatElec_CTA := 			ETOR9_Def_Alim_BatElec_CTA;
	E_Marche_BatElec_CTA := 			ETOR13_Marche_BatElec_CTA;
	E_Def_Humi_CTA := 					ETOR5_Def_Humi_CTA;
	E_Service_Humi_CTA := 				ETOR4_Service_Humi_CTA;
	E_Pressostat_Secu := 				ETOR11_Pressostat_Secu;
	E_Thermostat_Secu :=				ETOR12_Thermostat_Secu;

	STOR4_Cmd_BatElec_CTA := 			S_Cmd_BatElec_CTA;
	Var_BOOL_Bidon := 					S_Cmd_Humi_CTA;

	SAN5_Cons_V3V_Froid_CTA := 			S_Cons_V3V_Froid_CTA;
	SAN2_Cons_MotRep_CTA := 			S_Cons_MotRep_CTA;
	SAN3_Cons_MotSouf_CTA := 			S_Cons_MotSouf_CTA;
	SAN4_Cons_BatElec_CTA := 			S_Cons_BatElec_CTA;
	SAN1_Cons_Humi_CTA := 				S_Cons_Humi_CTA;

END_PROGRAM

// ---- POUs/a3_Ecriture_Bit.TcPOU
PROGRAM a3_Ecriture_Bit
VAR
	TP_RAZ_Marche_Manu: TP;
	TP_RAZ_Stop_Manu: TP;
	TP_RAZ_Depollution: TP;
	TP_RAZ_Valid: TP;
	TP_RAZ_Pause: TP;
	TP_RAZ_Valid_Recette: TP;
	TP_RAZ_Marche_Auto: TP;
	TP_RAZ_Stop_Auto: TP;
	TP_RAZ_Rearm: TP;
	TP_RAZ_Enr_Recette: TP;
	TP_RAZ_MAL: TP;
	TP_RAZ_FWCGV: TP;
	TP_RAZ_FWCPV: TP;
END_VAR

(**********************************************Gestion des RAZ des Bits d'écriture de l'IHM et GTC*)
TP_RAZ_Marche_Manu(IN:= %MX17422.0, PT:= T#1S);
%MX17422.0 := (SEL(%MX17422.0, %MX17422.0, FALSE) OR TP_RAZ_Marche_Manu.Q);

TP_RAZ_Stop_Manu(IN:= %MX17422.1, PT:= T#1s);
%MX17422.1 := (SEL(%MX17422.1, %MX17422.1, FALSE) OR TP_RAZ_Stop_Manu.Q);

TP_RAZ_Depollution(IN:= %MX17422.2, PT:= T#1s);
%MX17422.2 := (SEL(%MX17422.2, %MX17422.2, FALSE) OR TP_RAZ_Depollution.Q);

TP_RAZ_Valid(IN:= %MX17422.6, PT:= T#2s);
%MX17422.6 := (SEL(%MX17422.6, %MX17422.6, FALSE) OR TP_RAZ_Valid.Q);

TP_RAZ_Pause(IN:= %MX17422.7, PT:= T#1s);
%MX17422.7 := (SEL(%MX17422.7, %MX17422.7, FALSE) OR TP_RAZ_Pause.Q);

TP_RAZ_Valid_Recette(IN:= %MX17422.9, PT:= T#5s);
%MX17422.9 := (SEL(%MX17422.9, %MX17422.9, FALSE) OR TP_RAZ_Valid_Recette.Q);

TP_RAZ_Marche_Auto(IN:= %MX17422.10, PT:= T#5s);
%MX17422.10 := (SEL(%MX17422.10, %MX17422.10, FALSE) OR TP_RAZ_Marche_Auto.Q);

TP_RAZ_Stop_Auto(IN:= %MX17422.11, PT:= T#1s);
%MX17422.11 := (SEL(%MX17422.11, %MX17422.11, FALSE) OR TP_RAZ_Stop_Auto.Q);

TP_RAZ_Rearm(IN:= %MX17422.12, PT:= T#1s);
%MX17422.12 := (SEL(%MX17422.12, %MX17422.12, FALSE) OR TP_RAZ_Rearm.Q);

TP_RAZ_Enr_Recette(IN:= %MX17422.13, PT:= T#5s);
%MX17422.13 := (SEL(%MX17422.13, %MX17422.13, FALSE) OR TP_RAZ_Enr_Recette.Q);

TP_RAZ_MAL(IN:= %MX17434.7, PT:= T#1S);
%MX17434.7 := (SEL(%MX17434.7, %MX17434.7, FALSE) OR TP_RAZ_MAL.Q);

TP_RAZ_FWCGV(IN:= %MX17438.2, PT:= T#2S);
%MX17438.2 := (SEL(%MX17438.2, %MX17438.2, FALSE) OR TP_RAZ_FWCGV.Q);

TP_RAZ_FWCPV(IN:= %MX17438.4, PT:= T#2s);
%MX17438.4 := (SEL(%MX17438.4, %MX17438.4, FALSE) OR TP_RAZ_FWCPV.Q);

(**********************************************Variable Ecr_Bit_Cmd_IHM1*) (*Adresse Modbus GTC : 20999*)
(*Bit ecriture gestion recette*)
Start_Mode_Manu := 					Start_Mode_Manu; (*Impultion*)
Reset_Mode_Manu := 					Reset_Mode_Manu; (*Impultion*)
Start_Etat_Depollution := 			Start_Etat_Depollution; (*Impultion*)
Start_Etat_Nettoyage := 			Start_Etat_Nettoyage;
Activation_Ecl := 					Activation_Ecl;
Choix_Langue :=						Choix_Langue;
Valid_Texte := 						Valid_Texte; (*Impultion*)
Bp_Pause :=							Bp_Pause; (*Impultion*)
Detail_Nom_Recette_Mode :=			Detail_Nom_Recette_Mode;
Validation_Recette_Auto :=			Validation_Recette_Auto; (*Impultion*)
Start_Recette_Mode_Auto :=			Start_Recette_Mode_Auto; (*Impultion*)
Reset_Mode_Auto := 					Reset_Mode_Auto; (*Impultion*)
Cmd_Rearmement :=					Cmd_Rearmement; (*Impultion*)
Cmd_Enr_Recette :=					Cmd_Enr_Recette; (*Impultion*)
Cmd_Mode_Maintenance :=				Cmd_Mode_Maintenance;

(**********************************************GESTION DES OPTIONS*)

(*Option types de cabine*)
Option_Cabine_Seche := 				Option_Cabine_Seche; (*Adresse Modbus GTC : 21001 bit 0*)
Option_Cabine_Humide := 			Option_Cabine_Humide; (*Adresse Modbus GTC : 21001 bit 1*)
Option_Cabine_Climatique := 		Option_Cabine_Climatique; (*Adresse Modbus GTC : 21002 bit 15*)

(*Option actionneurs*)
Option_Douche := 					Option_Douche; (*Adresse Modbus GTC : 21001 bit 2*)
Option_Lavabo := 					Option_Lavabo; (*Adresse Modbus GTC : 21001 bit 3*)
Option_Douchette := 				Option_Douchette; (*Adresse Modbus GTC : 21001 bit 4*)
Option_NEP := 						Option_NEP; (*Adresse Modbus GTC : 21002 bit 14*)
Option_Prise :=						Option_Prise; (*Adresse Modbus GTC : 21001 bit 5*)
Option_WC_GV :=						Option_WC_GV; (*Adresse Modbus GTC : 21000 bit 0*)
Option_WC_PV :=						Option_WC_PV; (*Adresse Modbus GTC : 21000 bit 1*)
Option_RegSouf_Ultrason := 			Option_RegSouf_Ultrason; (*Adresse Modbus GTC : 21002 bit 12*)
Option_Reg_Etanche_Ext := 			Option_Reg_Etanche_Ext; (*Adresse Modbus GTC : 21002 bit 0*)
Option_V3V_EauMitig :=				Option_V3V_EauMitig; (*Adresse Modbus GTC : 21001 bit 8*)
Option_RegExt_Ultrason := 			Option_RegExt_Ultrason; (*Adresse Modbus GTC : 21002 bit 13*)
Option_Reg_Etanche_Souf := 			Option_Reg_Etanche_Souf; (*Adresse Modbus GTC : 21002 bit 7*)
Option_Bas_Debit :=					Option_Bas_Debit; (*Adresse Modbus GTC : 21001 bit 10*)
Option_Batt_Elec := 				Option_Batt_Elec; (*Adresse Modbus GTC : 21002 bit 3*)
Option_Mot_ByPass := 				Option_Mot_ByPass; (*Adresse Modbus GTC : 21002 bit 4*)
Option_Pompe_De_Relevage :=			Option_Pompe_De_Relevage; (*Adresse Modbus GTC : 21001 bit 13*)

(*Option capteurs*)
Option_Debitmetre_Douche := 		Option_Debitmetre_Douche; (*Adresse Modbus GTC : 21002 bit 1*)
Option_Debitmetre_Lavabo := 		Option_Debitmetre_Lavabo; (*Adresse Modbus GTC : 21002 bit 2*)
Option_Sonde_Temp_Hygro_Amb := 		Option_Sonde_Temp_Hygro_Amb; (*Adresse Modbus GTC : 21001 bit 11*)
Option_Capteur_Press_Cab := 		Option_Capteur_Press_Cab; (*Adresse Modbus GTC : 21002 bit 6*)
Option_Sonde_Temp_EauMitig :=		Option_Sonde_Temp_EauMitig; (*Adresse Modbus GTC : 21001 bit 7*)
Option_Press_SoufExt_General  :=	Option_Press_SoufExt_General; (*Adresse Modbus GTC : 21000 bit 2*)
Option_Temp_Batterie_EG  :=			Option_Temp_Batterie_EG; (*Adresse Modbus GTC : 21000 bit 3*)
Option_Sonde_Temp_Amb :=			Option_Sonde_Temp_Amb; (*Adresse Modbus GTC : 21001 bit 12*)
Option_Contact_Porte := 			Option_Contact_Porte; (*Adresse Modbus GTC : 21002 bit 0*)
Option_Niveau_Haut_Douche :=		Option_Niveau_Haut_Douche; (*Adresse Modbus GTC : 21001 bit 14*)
Option_Niveau_Haut_Lavabo :=		Option_Niveau_Haut_Lavabo; (*Adresse Modbus GTC : 21001 bit 15*)
Option_Defaut_Prise_Elec := 		Option_Defaut_Prise_Elec; (*Adresse Modbus GTC : 21002 bit 10*)

(*Option communication*)
Option_InterCom := 					Option_InterCom; (*Adresse Modbus GTC : 21001 bit 6*)
Option_Com_RegSouf_Ultrason := 		Option_Com_RegSouf_Ultrason; (*Adresse Modbus GTC : 21002 bit 5*)
Option_Com_RegExt_Ultrason := 		Option_Com_RegExt_Ultrason; (*Adresse Modbus GTC : 21002 bit 0*)

(*Option régulations*)
Option_Regul_Deb_Ou_Press := 		Option_Regul_Deb_Ou_Press; (*Adresse Modbus GTC : 21002 bit 8*)
Option_Regul_Temp_Eau :=			Option_Regul_Temp_Eau; (*Adresse Modbus GTC : 21001 bit 9*)

(**********************************************Variable Ecr_Bit_Cmd_IHM5*) (*Adresse Modbus GTC : 21003*)
(*Gestion des forçages*)
EF_Cmd_PC_Cab := 					EF_Cmd_PC_Cab;
EF_Cmd_Vanne_Alim_Douche := 		EF_Cmd_Vanne_Alim_Douche;
EF_Cmd_Vanne_Alim_Douchette := 		EF_Cmd_Vanne_Alim_Douchette;
EF_Cmd_Vanne_Alim_Lavabo := 		EF_Cmd_Vanne_Alim_Lavabo;
EF_Cmd_Vanne_Vid_Douche := 			EF_Cmd_Vanne_Vid_Douche;
EF_Cmd_Vanne_Vid_Lavabo :=			EF_Cmd_Vanne_Vid_Lavabo;
EF_Cmd_ElectroValve_Alim_Douche := 	EF_Cmd_ElectroValve_Alim_Douche;
EF_Cmd_ElectroValve_Alim_Lavabo :=	EF_Cmd_ElectroValve_Alim_Lavabo;
EF_Cons_Registre_Extraction :=		EF_Cons_Registre_Extraction;
EF_Cons_Registre_Soufflage :=		EF_Cons_Registre_Soufflage;
EF_Vanne_Souf_Bas_Deb :=			EF_Vanne_Souf_Bas_Deb;
EF_Vanne_Ext_Bas_Deb :=				EF_Vanne_Ext_Bas_Deb;
EF_Cons_Reg_Etanche_Ext :=			EF_Cons_Reg_Etanche_Ext;
EF_Cmd_Reg_Etanche_Souf :=			EF_Cmd_Reg_Etanche_Souf;
EF_Cons_V3V_Eau_Mitig :=			EF_Cons_V3V_Eau_Mitig;
EF_Vanne_Alim_NEP :=				EF_Vanne_Alim_NEP;
EF_Cons_V3V_Bat_Froid_CTA := 		EF_Cons_V3V_Bat_Froid_CTA;
EF_Cmd_Verin_WC_GV := 				EF_Cmd_Verin_WC_GV;
EF_Cmd_Verin_WC_PV := 				EF_Cmd_Verin_WC_PV;

(**********************************************Variable Ecr_Bit_Cmd_IHM6*) (*Adresse Modbus GTC : 21004*)
(*Gestion des forçages*)
F_Cmd_PC_Cab := 					F_Cmd_PC_Cab;
F_Cmd_Vanne_Alim_Douche := 			F_Cmd_Vanne_Alim_Douche;
F_Cmd_Vanne_Alim_Douchette := 		F_Cmd_Vanne_Alim_Douchette;
F_Cmd_Vanne_Alim_Lavabo := 			F_Cmd_Vanne_Alim_Lavabo;
F_Cmd_Vanne_Vid_Douche := 			F_Cmd_Vanne_Vid_Douche;
F_Cmd_Vanne_Vid_Lavabo :=			F_Cmd_Vanne_Vid_Lavabo;
F_Cmd_ElectroValve_Alim_Douche := 	F_Cmd_ElectroValve_Alim_Douche;
F_Cmd_ElectroValve_Alim_Lavabo :=	F_Cmd_ElectroValve_Alim_Lavabo;
F_Vanne_Souf_Bas_Deb :=				F_Vanne_Souf_Bas_Deb;
F_Vanne_Ext_Bas_Deb :=				F_Vanne_Ext_Bas_Deb;
F_Cmd_Reg_Etanche_Souf :=			F_Cmd_Reg_Etanche_Souf;
F_Vanne_Alim_NEP :=					F_Vanne_Alim_NEP;
F_Cmd_Verin_WC_GV := 				F_Cmd_Verin_WC_GV; (*Impultion*)
F_Cmd_Verin_WC_PV := 				F_Cmd_Verin_WC_PV; (*Impultion*)

(**********************************************Variable Ecr_Bit_Cmd_IHM7*) (*Adresse Modbus GTC : 21005*)
(*Bit horodatage*)
Sel_Lundi := 						Sel_Lundi;
Sel_Mardi := 						Sel_Mardi;
Sel_Mercredi := 					Sel_Mercredi;
Sel_Jeudi := 						Sel_Jeudi;
Sel_Vendredi := 					Sel_Vendredi;
Sel_Samedi :=						Sel_Samedi;
Sel_Dimanche := 					Sel_Dimanche;
StartMiseALheure  := 				StartMiseALheure; (*Impultion*)

END_PROGRAM

// ---- POUs/a4_Lecture_Bit.TcPOU
PROGRAM a4_Lecture_Bit
VAR
END_VAR

(**********************************************Variable Lect_Bit_IHM1*) (*Adresse Modbus GTC : 21009*)
(*Gestion des défauts*)
%MX17442.0 := Defaut_Debordement_Douche;
%MX17442.1 := Defaut_Debordement_Lavabo;
%MX17442.2 := Defaut_Discord_Deb_Eau_Douche;
%MX17442.3 := Defaut_Discord_Deb_Eau_Lavabo;
%MX17442.4 := Defaut_Discord_PC_Cab;
%MX17442.5 := Def_Discord_Alim_Prise;
%MX17442.6 := Def_Prise_Porte_Ouverte;
%MX17442.7 := Defaut_Pompe_Relevage;
%MX17442.8 := Defaut_Porte_Ouverte;
%MX17442.9 := Defaut_Com_Dalcnet;
%MX17442.10 := Defaut_Com_Vanne_Thermo;
%MX17442.11 := Defaut_Com_Vanne_General;
%MX17442.12 := Defaut_Com_Client;
%MX17442.13 := Defaut_Discord_Vanne_Vid_Douche_Ouv;
%MX17442.14 := Defaut_Discord_Vanne_Vid_Douche_Ferm;
%MX17442.15 := Defaut_Discord_Vanne_Vid_Lavabo_Ouv;

(**********************************************Variable Lect_Bit_IHM2*) (*Adresse Modbus GTC : 21010*)
(*Gestion des défauts*)
%MX17444.0 := Defaut_Discord_Vanne_Vid_Lavabo_Ferm;
%MX17444.1 := Defaut_Discord_Vanne_Alim_Douche_Ouv;
%MX17444.2 := Defaut_Discord_Vanne_Alim_Douche_Ferm;
%MX17444.3 := Defaut_Discord_Vanne_Alim_Lavabo_Ouv;
%MX17444.4 := Defaut_Discord_Vanne_Alim_Lavabo_Ferm;
%MX17444.5 := Defaut_Discord_Vanne_Alim_Douchette_Ouv;
%MX17444.6 := Defaut_Discord_Vanne_Alim_Douchette_Ferm;
%MX17444.7 := Defaut_Discord_Deb_Ext;
%MX17444.8 := Defaut_Discord_Deb_Souf;
%MX17444.9 := Defaut_Discord_Reg_Souf_Ferm;
%MX17444.10 := Defaut_Discord_Reg_Ext_Ferm;
%MX17444.11 := Defaut_Klixon_BattElec;
%MX17444.12 := Defaut_Differentiel_Prise_Elec;
%MX17444.13 := Defaut_Discord_Vanne_Souf_Bas_Deb_Ouv;
%MX17444.14 := Defaut_Discord_Vanne_Souf_Bas_Deb_Ferm;
%MX17444.15 := Defaut_Discord_Vanne_Ext_Bas_Deb_Ouv;

(**********************************************Variable Lect_Bit_IHM7*) (*Adresse Modbus GTC : 21015*)
(*Gestion des défauts*)
%MX17454.0 := Defaut_Discord_Vanne_Ext_Bas_Deb_Ferm;
%MX17454.1 := Defaut_Discord_Reg_Etanche_Ext;
%MX17454.2 := Defaut_Discord_Regul_Press_Cab;
%MX17454.3 :=Defaut_Com_Reg_Souf ;
%MX17454.4 := Defaut_Com_Reg_Ext;
%MX17454.5 := Defaut_Ensemble_Bas_Debit;
%MX17454.6 := Defaut_Ensemble_Bypass;
%MX17454.7 := Defaut_Sonde_Press_Cabine;
%MX17454.8 := Defaut_Sonde_Temp_Cabine;
%MX17454.9 := Defaut_Sonde_Hygro_Cabine;
%MX17454.10 := Defaut_Sonde_Temp_Eau_Mitig;
%MX17454.11 := Defaut_Discord_Vanne_Alim_NEP_Ouv;
%MX17454.12 := Defaut_Discord_Vanne_Alim_NEP_Ferm;

(**********************************************Variable Lect_Bit_IHM3*) (*Adresse Modbus GTC : 21011*)
(*configuration des Entrees et sorties tor*)
%MX17446.0 := E_Info_Niveau_Haut_Douche;
%MX17446.1 := E_Info_Niveau_Haut_Lavabo;
%MX17446.2 := E_Info_Contact_Porte;
%MX17446.3 := E_Info_PC_Cab;
%MX17446.4 := E_Etat_Evac_SaniDouche;
%MX17446.5 := E_Vanne_Alim_Douche_Ouv;
%MX17446.6 := E_Vanne_Alim_Douche_Ferm;
%MX17446.7 := E_Vanne_Alim_Douchette_Ouv;
%MX17446.8 := E_Vanne_Alim_Douchette_Ferm;
%MX17446.9 := E_Vanne_Alim_Lavabo_Ouv;
%MX17446.10 := E_Vanne_Alim_Lavabo_Ferm;
%MX17446.11 := E_Vanne_Vidange_Douche_Ouv;
%MX17446.12 := E_Vanne_Vidange_Douche_Ferm;
%MX17446.13 := E_Vanne_Vidange_Lavabo_Ouv;
%MX17446.14 := E_Vanne_Vidange_Lavabo_Ferm;
%MX17446.15 := S_Cmd_PC_Cab;

(**********************************************Variable Lect_Bit_IHM4*) (*Adresse Modbus GTC : 21012*)
(*configuration des Entrees et sorties tor*)
%MX17448.0 := S_Cmd_Vanne_Alim_Douche;
%MX17448.1 := S_Cmd_Vanne_Alim_Douchette;
%MX17448.2 := S_Cmd_Vanne_Alim_Lavabo;
%MX17448.3 := S_Cmd_Vanne_Vid_Douche;
%MX17448.4 := S_Cmd_Vanne_Vid_Lavabo;
%MX17448.5 := S_Cmd_ElectroValve_Alim_Douche;
%MX17448.6 := S_Cmd_ElectroValve_Alim_Lavabo;
%MX17448.7 := S_Cmd_Vanne_Souf_Bas_Deb;
%MX17448.8 := S_Cmd_Vanne_Ext_Bas_Deb;
%MX17448.9 := E_Vanne_Souf_Bas_Deb_Ouv;
%MX17448.10 := E_Vanne_Souf_Bas_Deb_Ferm;
%MX17448.11 := E_Vanne_Ext_Bas_Deb_Ouv;
%MX17448.12 := E_Vanne_Ext_Bas_Deb_Ferm;
%MX17448.13 := E_Defaut_Prise_Elec;
%MX17448.14 := E_Info_Klixon_BattElec;
%MX17448.15 := S_Cmd_Reg_Etanche_Souf;

(**********************************************Variable Lect_Bit_IHM8*) (*Adresse Modbus GTC : 21016*)
(*configuration des Entrees et sorties tor*)
%MX17456.0 :=	E_Vanne_Alim_NEP_Ouv;
%MX17456.1 := 	E_Vanne_Alim_NEP_Ferm;
%MX17456.2 :=	S_Cmd_Vanne_NEP;
%MX17456.3 :=	S_Cmd_Appli_Verin_WC_GV;
%MX17456.4 :=	S_Cmd_Appli_Verin_WC_PV;

(**********************************************Variable Lect_Bit_IHM5*) (*Adresse Modbus GTC : 21013*)
(*Bit lecture gestion recette et état de la cabine*)
%MX17450.0 := Mode_Cabine_Eclairage;
%MX17450.1 := Mode_Cabine_Libre;
%MX17450.2 := Mode_Cabine_Manuel;
%MX17450.3 := Mode_Cabine_Automatique;
%MX17450.4 := Mode_Cabine_Depollution;
%MX17450.5 := Mode_Cabine_Nettoyage;
%MX17450.6 := Mode_Evaluation;
%MX17450.7 := Mode_Neutre;
%MX17450.8 := Mode_Cabine_Defaut;
%MX17450.9 := Mode_Maintenance;

(**********************************************Variable Lect_Bit_IHM6*) (*Adresse Modbus GTC : 21014*)
(*Bit lecture gestion recette et état de la cabine*)
%MX17452.0 := Statut_Pause_Force;
%MX17452.1 := Attente_Reset_Pause;
%MX17452.2 := Comande_Pause;
%MX17452.3 := Condi_Affich_Etape_Suiv;
%MX17452.4 := Condi_Affich_Rearm;
%MX17452.5 := Enable_PID_Bas_Deb_Ext;
%MX17452.6 := Enable_PID_Press_Cab;
%MX17452.7 := Enable_PID_Temp_Eau_Mitig;

(*Mise à zéro des défaut si mode maintenance*)
IF(Cmd_Mode_Maintenance)
	THEN
	%MW17442 := 0;
	%MW17444 := 0;
	%MW17454 := 0;
	%MW17458 := 0;
END_IF;

(**********************************************Variable Lect_Bit_IHM9*) (*Adresse Modbus GTC : 21017*)
(*Bit lecture gestion enceinte climatique*)
%MX17458.0 := Defaut_MotRep_CTA;
%MX17458.1 := Defaut_MotSouf_CTA;
%MX17458.2 := Defaut_Hygrostat_CTA;
%MX17458.3 := Defaut_Alim_BatElec_CTA;
%MX17458.4 := Defaut_Humi_CTA;
%MX17458.5 := Defaut_Regul_Temp;
%MX17458.6 := Defaut_Regul_Hygro;
%MX17458.7 := S_Cmd_BatElec_CTA;
%MX17458.8 := S_Cmd_Humi_CTA;
%MX17458.9 := E_Pressostat_Secu;
%MX17458.10 := E_Marche_BatElec_CTA;
%MX17458.11 := E_Service_Humi_CTA;

(**********************************************Variable Lect_Bit_IHM10*) (*Adresse Modbus GTC : 21018*)
%MX17460.0 := GVL_RegTROX.RegSouf_GD_FCVT01_DefCom;
%MX17460.1 := GVL_RegTROX.RegSouf_GD_FCVT01_Def_DiscordDeb;
%MX17460.2 := GVL_RegTROX.RegSouf_PD_FCVT02_DefCom;
%MX17460.3 := GVL_RegTROX.RegSouf_PD_FCVT02_Def_DiscordDeb;
%MX17460.4 := GVL_RegTROX.RegSouf_Cabine_FCVT03_DefCom;
%MX17460.5 := GVL_RegTROX.Reg_Bypass_FCVT04_DefCom;
%MX17460.6 := GVL_RegTROX.Reg_Bypass_FCVT04_Def_DiscordDeb;
%MX17460.7 := GVL_RegTROX.RegSouf_CabGD_FCVT05_DefCom;
%MX17460.8 := GVL_RegTROX.RegSouf_CabGD_FCVT05_Def_DiscordDeb;
%MX17460.9 := GVL_RegTROX.RegSouf_CabPD_FCVT06_DefCom;
%MX17460.10 := GVL_RegTROX.RegSouf_CabPD_FCVT06_Def_DiscordDeb;
%MX17460.11 := GVL_RegTROX.RegRep_FCVT07_DefCom;
%MX17460.12 := Defaut_Discord_Souf_CTA;
%MX17460.13 := Defaut_Thermostat_Secu;
%MX17460.14 := Defaut_Sonde_Temp_Souf;

END_PROGRAM

// ---- POUs/a5_Ecriture_InterCom.TcPOU
PROGRAM a5_Ecriture_InterCom
VAR
	Position_Soufflage: REAL;
	Position_Extraction: REAL;
	Mesure_Debit_Souf: REAL;
	Mesure_Debit_Ext: REAL;
	Com_Debit_Ext: REAL;
	Dmd_Mise_En_Temp: BOOL;
END_VAR

Temperature_Cabine := Tab_MES_Sonde_Temp_Amb.R_MesCor;
Hygrometrie_Cabine := Tab_MES_Sonde_Hygro_Amb.R_MesCor;
Position_Soufflage := Posi_Relative_Reg_Souf / 100.0;
Position_Extraction := Cons_Actionneur_Reg_Etanche_Ext;
Com_Debit_Ext := Debit_Relative_Reg_Souf;
Mesure_Debit_Souf := Tab_MES_Sonde_Gros_Debit_Soufflage.R_MesCor;
Mesure_Debit_Ext := Tab_MES_Sonde_Gros_Debit_Extraction.R_MesCor;
Dmd_Mise_En_Temp := E_Vanne_Alim_Lavabo_Ouv OR E_Vanne_Alim_Douche_Ouv OR S_Cmd_ElectroValve_Alim_Lavabo OR S_Cmd_ElectroValve_Alim_Douche;

(**********************************************Gestion écriture inter com*)
Tab_Com_Send[0] := 		Temperature_Cabine;
Tab_Com_Send[1] := 		Hygrometrie_Cabine;
Tab_Com_Send[2] := 		FCV_02_soufflage.Cons_Pos_Dem;
Tab_Com_Send[3] := 		FCV_01_extraction.Cons_Pos_Dem;
Tab_Com_Send[4] := 		Sel_Etats_Cabine;
Tab_Com_Send[5] := 		Position_Extraction;
Tab_Com_Send[6] := 		Position_Soufflage;
Tab_Com_Send[7] := 		Mesure_Debit_Souf;
Tab_Com_Send[8] := 		Mesure_Debit_Ext;
Tab_Com_Send[9] := 		BOOL_TO_REAL(Dmd_Mise_En_Temp);
Tab_Com_Send[10] := 	BOOL_TO_REAL(Defaut_Sonde_Temp_Cabine);
Tab_Com_Send[11] := 	Mode_Manu.Numero_Mode;
Tab_Com_Send[12] := 	BOOL_TO_REAL(Mode_Cabine_Depollution OR Mode_Auto.Mode_10);

END_PROGRAM

// ---- POUs/a6_Lecture_InterCom.TcPOU
PROGRAM a6_Lecture_InterCom
VAR
	Cons_Temp_Eau_General: REAL;
END_VAR

(**********************************************Gestion lecture inter com*)
MES_Temp_Eau_Mitige_General := Tab_Com_Receive[0];
Cons_Temp_Eau_General		:= Tab_Com_Receive[1];

END_PROGRAM

// ---- POUs/b_SCL_Mesures.TcPOU
PROGRAM b_SCL_Mesures
VAR
(*Mesure sonde de température d'ambiance*)
	Objet_Sonde_Temp_Amb			:Objet_Sonde_V1;
(*Mesure sonde d'hygrométrie d'ambiance*)
	Objet_Sonde_Hygro_Amb 			:Objet_Sonde_V1;
(*Mesure sonde de température d'eau mitigée*)
	Objet_Sonde_Temp_Eau_Mitig		:Objet_Sonde_V1;
(*Mesure Gros débit de soufflage*)
	Objet_Sonde_Gros_Debit_Soufflage 	:Objet_Sonde_V1;
	TON_F1: TON;
	Filtre_V1_Soufflage: Filtre_V1;
(*Mesure Gros débit d'extraction*)
	Objet_Sonde_Gros_Debit_Extraction 	:Objet_Sonde_V1;
	TON_F2: TON;
	Filtre_V1_Extraction: Filtre_V1;
(*Mesure Petit débit d'extraction*)
	Objet_Sonde_Petit_Debit_Extraction 	:Objet_Sonde_V1;
	TON_F3: TON;
	E_Sonde_Petit_Debit_Extraction_1 :INT;
	Filtre_V1_BasDebit: Filtre_V1;
	Calcul_1: REAL;
	Calcul_2: REAL;
	Calcul_3: REAL;
	Calcul_4: REAL;
	TON_PD :TON;
(*Mesure débit d'eau d'alimentation de la douche*)
	Objet_Sonde_Debit_Alim_Douche 	:Objet_Sonde_V1;
	TON_F4: TON;
	MES_MIN_Douche: REAL;
(*Mesure débit d'eau d'alimentation du lavabo*)
	Objet_Sonde_Debit_Alim_Lavabo	:Objet_Sonde_V1;
	TON_F5: TON;
	MES_MIN_Lavabo: REAL;
(*Mesure sonde de pression de la cabine*)
	Objet_Sonde_Press_Cab			:Objet_Sonde_V1;
(*Mesure Pression ByPass*)
	Objet_Sonde_Press_Bypass 	:Objet_Sonde_V1;
	TON_F6: TON;
	E_Sonde_Pression_ByPass_1 :INT;
	Filtre_V1_ByPass: Filtre_V1;
	Calcul_5: REAL;
	Calcul_6: REAL;
	TON_P1 :TON;
(*Mesure retour d'information du registre étanche extraction*)
	SCL_Pos_Reg_Etanche_Ext	:SCL;
(*Mesure sonde de pression de soufflage general*)
	Objet_Sonde_V1_Press_Souf: Objet_Sonde_V1;
(*Mesure sonde de pression d'extraction general*)
	Objet_Sonde_V1_Press_Ext: Objet_Sonde_V1;
(*Mesure sonde de température batterie eau glacée*)
	Objet_Sonde_Temp_Batt_EG		:Objet_Sonde_V1;
(*Mesure sonde de température de soufflage*)
	Objet_Sonde_Temp_Souf			:Objet_Sonde_V1;
END_VAR

(**********************************************Mesure sonde de température d'ambiance*)
IF(Option_Sonde_Temp_Hygro_Amb OR Option_Sonde_Temp_Amb) (*Gestion des options*)
	THEN	E_Sonde_Temp_Amb := E_Sonde_Temp_Amb;
	ELSE	E_Sonde_Temp_Amb := 0;
END_IF;

(*Objet sonde*)
Objet_Sonde_Temp_Amb(
	Mesure_EAN:= INT_TO_REAL(E_Sonde_Temp_Amb),
	Enable_Alarme:= FALSE,
	Status_DEF_EAN:= FALSE,
	Tempo_AL:= T#60s,
	Hyst_AL:= 1.0,
	EAN_MIN:= 0.0,
	EAN_MAX:= 32767.0,
	MES_MIN:= -20.0,
	MES_MAX:= 80.0,
	Filtre_Actif:= FALSE,
	Temps_Echantillonage:= T#1s,
	Tab_Sonde:= Tab_MES_Sonde_Temp_Amb);
Tab_MES_Sonde_Temp_Amb.R_MesCor := Tab_MES_Sonde_Temp_Amb.R_MesCor;

(**********************************************Mesure sonde d'hygrométrie d'ambiance*)
IF(Option_Sonde_Temp_Hygro_Amb) (*Gestion des options*)
	THEN	E_Sonde_Hygro_Amb := E_Sonde_Hygro_Amb;
	ELSE	E_Sonde_Hygro_Amb := 0;
END_IF;

(*Objet sonde*)
Objet_Sonde_Hygro_Amb(
	Mesure_EAN:= INT_TO_REAL(E_Sonde_Hygro_Amb),
	Enable_Alarme:= FALSE,
	Status_DEF_EAN:= FALSE,
	Tempo_AL:= T#60s,
	Hyst_AL:= 5.0,
	EAN_MIN:= 0.0,
	EAN_MAX:= 32767.0,
	MES_MIN:= 0.0,
	MES_MAX:= 100.0,
	Filtre_Actif:= FALSE,
	Temps_Echantillonage:= T#1s,
	Tab_Sonde:= Tab_MES_Sonde_Hygro_Amb);
Tab_MES_Sonde_Hygro_Amb.R_MesCor := Tab_MES_Sonde_Hygro_Amb.R_MesCor;

(**********************************************Mesure sonde de température d'eau mitigée*)
IF(Option_Sonde_Temp_EauMitig) (*Gestion des options*)
	THEN	E_Sonde_Temp_Eau_Mitig := E_Sonde_Temp_Eau_Mitig;
	ELSE	E_Sonde_Temp_Eau_Mitig := 0;
END_IF;

(*Objet sonde*)
Objet_Sonde_Temp_Eau_Mitig(
	Mesure_EAN:= INT_TO_REAL(E_Sonde_Temp_Eau_Mitig),
	Enable_Alarme:= FALSE,
	Status_DEF_EAN:= FALSE,
	Tempo_AL:= T#60s,
	Hyst_AL:= 1.0,
	EAN_MIN:= 0.0,
	EAN_MAX:= 32767.0,
	MES_MIN:= -20.0,
	MES_MAX:= 80.0,
	Filtre_Actif:= FALSE,
	Temps_Echantillonage:= T#1s,
	Tab_Sonde:= Tab_MES_Sonde_Temp_Eau_Mitig);
Tab_MES_Sonde_Temp_Eau_Mitig.R_MesCor := Tab_MES_Sonde_Temp_Eau_Mitig.R_MesCor;

(**********************************************Mesure Gros débit de soufflage*)
IF(Option_RegSouf_Ultrason)
THEN
	(*Remise à zéro en cas de fermeture du registre et consigne inférieur pendant 30 secondes*)
	E_Sonde_Gros_Debit_Soufflage_1 := E_Sonde_Gros_Debit_Soufflage;
	TON_F1(IN:= (E_Sonde_Gros_Debit_Soufflage_1 < TOL_RAZ_MES_Deb_Souf), PT:= t#30s);
	IF(TON_F1.Q)
		THEN
		E_Sonde_Gros_Debit_Soufflage := 0;
	END_IF;

	(*Sélection de l'échelle maximum de mesure en fonction de la cabine seche ou humide / Humide : 662m3/h et seche : *)
	IF (Option_Cabine_Seche)
		THEN
		Mes_Out_Max := 579.0;
	END_IF;
	IF (Option_Cabine_Humide)
		THEN
		Mes_Out_Max := 579.0;
	END_IF;
ELSE
	TON_F1(IN:=FALSE);
	E_Sonde_Gros_Debit_Soufflage_1 := 0;
	E_Sonde_Gros_Debit_Soufflage := 0;
END_IF

(*Objet sonde*)
Objet_Sonde_Gros_Debit_Soufflage(
	Mesure_EAN:= INT_TO_REAL(E_Sonde_Gros_Debit_Soufflage),
	Enable_Alarme:= FALSE,
	Status_DEF_EAN:= FALSE,
	Tempo_AL:= T#60s,
	Hyst_AL:= 10.0,
	EAN_MIN:= 0.0,
	EAN_MAX:= 32767.0,
	MES_MIN:= 0.0,
	MES_MAX:= Mes_Out_Max,
	Filtre_Actif:= TRUE,
	Temps_Echantillonage:= T#500ms,
	Tab_Sonde:= Tab_MES_Sonde_Gros_Debit_Soufflage);
Tab_MES_Sonde_Gros_Debit_Soufflage.R_MesCor := Tab_MES_Sonde_Gros_Debit_Soufflage.R_MesCor;

(**********************************************Mesure Gros débit d'extraction*)
IF(Option_RegExt_Ultrason)
	THEN
	(*Remise à zéro en cas de fermeture du registre et consigne inférieur pendant 30 secondes*)
	E_Sonde_Gros_Debit_Extraction_1 := E_Sonde_Gros_Debit_Extraction;
	TON_F2(IN:= (E_Sonde_Gros_Debit_Extraction_1 < TOL_RAZ_MES_Deb_Ext), PT:= t#30s);
	IF(TON_F2.Q)
		THEN
		E_Sonde_Gros_Debit_Extraction := 0;
	END_IF;
ELSE
	TON_F2(IN:=FALSE);
	E_Sonde_Gros_Debit_Extraction_1 := 0;
	E_Sonde_Gros_Debit_Extraction := 0;
END_IF

(*Objet sonde*)
Objet_Sonde_Gros_Debit_Extraction(
	Mesure_EAN:= INT_TO_REAL(E_Sonde_Gros_Debit_Extraction),
	Enable_Alarme:= FALSE,
	Status_DEF_EAN:= FALSE,
	Tempo_AL:= T#60s,
	Hyst_AL:= 10.0,
	EAN_MIN:= 0.0,
	EAN_MAX:= 32767.0,
	MES_MIN:= 0.0,
	MES_MAX:= Mes_Out_Max,
	Filtre_Actif:= TRUE,
	Temps_Echantillonage:= T#500ms,
	Tab_Sonde:= Tab_MES_Sonde_Gros_Debit_Extraction);
Tab_MES_Sonde_Gros_Debit_Extraction.R_MesCor := Tab_MES_Sonde_Gros_Debit_Extraction.R_MesCor;

(**********************************************Mesure Petit débit d'extraction*)
IF(Option_Bas_Debit) (*Gestion des options*)
	THEN
	(*Remise à zéro en cas d'arrêt du moteur et consigne inférieur pendant 30 secondes*)
	E_Sonde_Petit_Debit_Extraction := E_Sonde_Petit_Debit_Extraction;
	E_Sonde_Petit_Debit_Extraction_1 := E_Sonde_Petit_Debit_Extraction;
	TON_F3(IN:= (E_Sonde_Petit_Debit_Extraction_1 < TOL_RAZ_MES_Petit_Deb), PT:= t#30s);
	IF( Arret_Petit_Debit  AND TON_F3.Q)
		THEN
		E_Sonde_Petit_Debit_Extraction := 0;
	END_IF;
ELSE
	TON_F3(IN:=FALSE);
	E_Sonde_Petit_Debit_Extraction_1 := 0;
	E_Sonde_Petit_Debit_Extraction := 0;
END_IF;

(*Objet sonde*)
Objet_Sonde_Petit_Debit_Extraction(
	Mesure_EAN:= INT_TO_REAL(E_Sonde_Petit_Debit_Extraction),
	Enable_Alarme:= FALSE,
	Status_DEF_EAN:= FALSE,
	Tempo_AL:= T#60s,
	Hyst_AL:= 0.0,
	EAN_MIN:= 1638, (*0,5V*)
	EAN_MAX:= 14745, (*4,5V*)
	MES_MIN:= 0.0,
	MES_MAX:= 300.0,
	Filtre_Actif:= FALSE,
	Temps_Echantillonage:= T#1s,
	Tab_Sonde:= Tab_MES_Sonde_Petit_Debit_Extraction);
Tab_MES_Sonde_Petit_Debit_Extraction.R_MesCor := Tab_MES_Sonde_Petit_Debit_Extraction.R_MesCor;

(**********************************************Mesure débit d'eau d'alimentation de la douche*)
IF(Option_Debitmetre_Douche) (*Gestion des options*)
	THEN
	E_Sonde_Debit_Alim_Douche := E_Sonde_Debit_Alim_Douche;
	MES_MIN_Douche := 0.0;
	(*Remise à zéro du débit d'eau en cas de fermeture de la vanne*)
	TON_F4(IN:= (NOT S_Cmd_ElectroValve_Alim_Douche), PT:= T#2S);
	IF(TON_F4.Q)
		THEN
		E_Sonde_Debit_Alim_Douche := 0;
		MES_MIN_Douche := 0.0;
	END_IF;
	ELSE
	TON_F4(IN:=FALSE);
	E_Sonde_Debit_Alim_Douche := 0;
	MES_MIN_Douche := 0.0;
END_IF;

(*Objet sonde*)
Objet_Sonde_Debit_Alim_Douche(
	Mesure_EAN:= INT_TO_REAL(E_Sonde_Debit_Alim_Douche) * Coef_Correction_DebitEau,
	Enable_Alarme:= FALSE,
	Status_DEF_EAN:= FALSE,
	Tempo_AL:= T#60s,
	Hyst_AL:= 0.0,
	EAN_MIN:= 0.0,
	EAN_MAX:= 32767.0,
	MES_MIN:= MES_MIN_Douche,
	MES_MAX:= 30.0,
	Filtre_Actif:= FALSE,
	Temps_Echantillonage:= T#1s,
	Tab_Sonde:= Tab_MES_Sonde_Debit_Alim_Douche);
Tab_MES_Sonde_Debit_Alim_Douche.R_MesCor := Tab_MES_Sonde_Debit_Alim_Douche.R_MesCor;

(**********************************************Mesure débit d'eau d'alimentation du lavabo*)
IF(Option_Debitmetre_Lavabo) (*Gestion des options*)
	THEN
	E_Sonde_Debit_Alim_Lavabo := E_Sonde_Debit_Alim_Lavabo;
	MES_MIN_Lavabo := 0.0;
	(*Remise à zéro du débit d'eau en cas de fermeture de la vanne*)
	TON_F5(IN:= (NOT S_Cmd_ElectroValve_Alim_Lavabo), PT:= t#2s);
	IF(TON_F5.Q)
		THEN
		E_Sonde_Debit_Alim_Lavabo := 0;
		MES_MIN_Lavabo := 0.0;
	END_IF;
	ELSE
	TON_F5(IN:=FALSE);
	E_Sonde_Debit_Alim_Lavabo := 0;
	MES_MIN_Lavabo := 0.0;
END_IF;

(*Objet sonde*)
Objet_Sonde_Debit_Alim_Lavabo(
	Mesure_EAN:= INT_TO_REAL(E_Sonde_Debit_Alim_Lavabo) * Coef_Correction_DebitEau,
	Enable_Alarme:= FALSE,
	Status_DEF_EAN:= FALSE,
	Tempo_AL:= T#60s,
	Hyst_AL:= 0.0,
	EAN_MIN:= 0.0,
	EAN_MAX:= 32767.0,
	MES_MIN:= MES_MIN_Lavabo,
	MES_MAX:= 30.0,
	Filtre_Actif:= FALSE,
	Temps_Echantillonage:= T#1s,
	Tab_Sonde:= Tab_MES_Sonde_Debit_Alim_Lavabo);
Tab_MES_Sonde_Debit_Alim_Lavabo.R_MesCor := Tab_MES_Sonde_Debit_Alim_Lavabo.R_MesCor;

(**********************************************Mesure sonde pression cabine*)
IF(Option_Capteur_Press_Cab) (*Gestion des options*)
	THEN	E_Sonde_Pression_Cabine := E_Sonde_Pression_Cabine;
	ELSE	E_Sonde_Pression_Cabine := 0;
END_IF;

(*Objet sonde*)
Objet_Sonde_Press_Cab(
	Mesure_EAN:= INT_TO_REAL(E_Sonde_Pression_Cabine),
	Enable_Alarme:= FALSE,
	Status_DEF_EAN:= FALSE,
	Tempo_AL:= T#60s,
	Hyst_AL:= 5.0,
	EAN_MIN:= 0.0,
	EAN_MAX:= 32767.0,
	MES_MIN:= -50.0,
	MES_MAX:= 50.0,
	Filtre_Actif:= FALSE,
	Temps_Echantillonage:= T#1s,
	Tab_Sonde:= Tab_MES_Sonde_Press_Cab);
Tab_MES_Sonde_Press_Cab.R_MesCor := Tab_MES_Sonde_Press_Cab.R_MesCor;

(**********************************************Mesure pression ByPass*)
IF(Option_Mot_ByPass) (*Gestion des options*)
	THEN
	(*Remise à zéro en cas d'arrêt du moteur et consigne inférieur pendant 30 secondes*)
	E_Sonde_Pression_ByPass := E_Sonde_Pression_ByPass;
	E_Sonde_Pression_ByPass_1 := E_Sonde_Pression_ByPass;
	TON_F6(IN:= (E_Sonde_Pression_ByPass_1 < TOL_RAZ_MES_Bypass), PT:= t#30s);
	IF(TON_F6.Q)
		THEN
		E_Sonde_Pression_ByPass := 0;
	END_IF;
	ELSE
	TON_F6(IN:=FALSE);
	E_Sonde_Pression_ByPass_1 := 0;
	E_Sonde_Pression_ByPass := 0;
END_IF;

(*Objet sonde*)
Objet_Sonde_Press_Bypass(
	Mesure_EAN:= INT_TO_REAL(E_Sonde_Pression_ByPass),
	Enable_Alarme:= FALSE,
	Status_DEF_EAN:= FALSE,
	Tempo_AL:= T#60s,
	Hyst_AL:= 0.0,
	EAN_MIN:= 0.0,
	EAN_MAX:= 16383.5,
	MES_MIN:= 0.0,
	MES_MAX:= 300.0,
	Filtre_Actif:= TRUE,
	Temps_Echantillonage:= T#1s,
	Tab_Sonde:= Tab_MES_Sonde_Press_ByPass);
Tab_MES_Sonde_Press_ByPass.R_MesCor := Tab_MES_Sonde_Press_ByPass.R_MesCor;

(**********************************************Mesure retour d'information du registre étanche extraction*)
IF(Option_Reg_Etanche_Ext) (*Gestion des options*)
	THEN	E_Retour_Pos_Reg_Etanche_Ext := E_Retour_Pos_Reg_Etanche_Ext;
	ELSE	E_Retour_Pos_Reg_Etanche_Ext := 0;
END_IF;

(*Mise à l'échelle de la mesure*)
SCL_Pos_Reg_Etanche_Ext(
	IN_INT:= E_Retour_Pos_Reg_Etanche_Ext,
	LIM_MIN_IN_REAL:= 6553.4,
	LIM_MAX_IN_REAL:= 32767.0,
	LIM_MIN_OUT_REAL:= 0.0,
	LIM_MAX_OUT_REAL:= 100.0,
	OUT_REAL=> MES_Pos_Reg_Etanche_Ext);

(**********************************************Mesure debit extraction bas débit*)
(*******Convertion de la pression en débit**********)
Calcul_1 := EXPT(Tab_MES_Sonde_Petit_Debit_Extraction.R_MesCor,4);
Calcul_2 := EXPT(Tab_MES_Sonde_Petit_Debit_Extraction.R_MesCor,3);
Calcul_3 := EXPT(Tab_MES_Sonde_Petit_Debit_Extraction.R_MesCor,2);
Calcul_4 := EXPT(Tab_MES_Sonde_Petit_Debit_Extraction.R_MesCor,1);
MES_Petit_Debit_m3h_Extraction :=  (-0.000000000905 * Calcul_1) + (0.00000114 * Calcul_2) - (0.000476 * Calcul_3) + (0.118 * Calcul_4) + 0.00303;

(*******Mise à zéro de la mesure en cas d'arrête*********)
TON_PD(IN:= (TON_F3.Q OR NOT Option_Bas_Debit), PT:= T#2s);
IF (TON_PD.Q)
	THEN
	MES_Petit_Debit_m3h_Extraction := 0.0;
	ELSE
	MES_Petit_Debit_m3h_Extraction := MES_Petit_Debit_m3h_Extraction;
END_IF;

